LIN {X 0,Y 227.107,Z 476.36,A -85,B 0,C 180,E1 -20579.094,E2 -20579.094} C_VEL
LIN {X 0,Y 226.995,Z 485.322,A -85,B 0,C 180,E1 -20580.664,E2 -20580.664} C_VEL
LIN {X 0,Y 226.013,Z 495.622,A -85,B 0,C 180,E1 -20582.704,E2 -20582.704} C_VEL
LIN {X 0,Y 223.02,Z 505.372,A -85,B 0,C 180,E1 -20584.828,E2 -20584.828} C_VEL
LIN {X 0,Y 220.277,Z 513.339,A -85,B 0,C 180,E1 -20586.998,E2 -20586.998} C_VEL
LIN {X 0,Y 217.787,Z 520.819,A -85,B 0,C 180,E1 -20589.579,E2 -20589.579} C_VEL
LIN {X 0,Y 215.866,Z 526.381,A -85,B 0,C 180,E1 -20591.988,E2 -20591.988} C_VEL
LIN {X 0,Y 214.036,Z 531.459,A -85,B 0,C 180,E1 -20594.775,E2 -20594.775} C_VEL
LIN {X 0,Y 212.725,Z 535.379,A -85,B 0,C 180,E1 -20597.604,E2 -20597.604} C_VEL
LIN {X 0,Y 211.981,Z 538.249,A -85,B 0,C 180,E1 -20600.463,E2 -20600.463} C_VEL
LIN {X 0,Y 211.672,Z 539.61,A -85,B 0,C 180,E1 -20602.373,E2 -20602.373} C_VEL
LIN {X 0,Y 211.57,Z 541.409,A -85,B 0,C 180,E1 -20604.285,E2 -20604.285} C_VEL
LIN {X 0,Y 211.515,Z 543.682,A -85,B 0,C 180,E1 -20606.194,E2 -20606.194} C_VEL
LIN {X 0,Y 211.604,Z 545.507,A -85,B 0,C 180,E1 -20608.101,E2 -20608.101} C_VEL
LIN {X 0,Y 211.672,Z 546.833,A -85,B 0,C 180,E1 -20610.004,E2 -20610.004} C_VEL
LIN {X 0,Y 211.55,Z 547.738,A -85,B 0,C 180,E1 -20611.908,E2 -20611.908} C_VEL
LIN {X 0,Y 211.496,Z 548.371,A -85,B 0,C 180,E1 -20615.725,E2 -20615.725} C_VEL
LIN {X 0,Y 212.119,Z 547.382,A -85,B 0,C 180,E1 -20619.54,E2 -20619.54} C_VEL
LIN {X 0,Y 213.535,Z 544.883,A -85,B 0,C 180,E1 -20623.324,E2 -20623.324} C_VEL
LIN {X 0,Y 215.163,Z 541.937,A -85,B 0,C 180,E1 -20626.123,E2 -20626.123} C_VEL
LIN {X 0,Y 217.434,Z 538.014,A -85,B 0,C 180,E1 -20628.862,E2 -20628.862} C_VEL
LIN {X 0,Y 220.15,Z 533.028,A -85,B 0,C 180,E1 -20631.542,E2 -20631.542} C_VEL
LIN {X 0,Y 223.777,Z 525.758,A -85,B 0,C 180,E1 -20634.594,E2 -20634.594} C_VEL
LIN {X 0,Y 227.652,Z 518.001,A -85,B 0,C 180,E1 -20637.092,E2 -20637.092} C_VEL
LIN {X 0,Y 231.21,Z 510.223,A -85,B 0,C 180,E1 -20639.104,E2 -20639.104} C_VEL
LIN {X 0,Y 234.36,Z 502.894,A -85,B 0,C 180,E1 -20640.654,E2 -20640.654} C_VEL
LIN {X 0,Y 236.711,Z 492.801,A -85,B 0,C 180,E1 -20642.823,E2 -20642.823} C_VEL
LIN {X 0,Y 238.09,Z 482.378,A -85,B 0,C 180,E1 -20644.888,E2 -20644.888} C_VEL
LIN {X 0,Y 238.492,Z 473.335,A -85,B 0,C 180,E1 -20646.63,E2 -20646.63} C_VEL
LIN {X 0,Y 238.102,Z 467.173,A -85,B 0,C 180,E1 -20647.913,E2 -20647.913} C_VEL
LIN {X 0,Y 237.355,Z 464.057,A -85,B 0,C 180,E1 -20648.702,E2 -20648.702} C_VEL
LIN {X 0,Y 234.077,Z 456.011,A -85,B 0,C 180,E1 -20651.356,E2 -20651.356} C_VEL
LIN {X 0,Y 231.692,Z 450.913,A -85,B 0,C 180,E1 -20653.28,E2 -20653.28} C_VEL
LIN {X 0,Y 229.388,Z 446.355,A -85,B 0,C 180,E1 -20655.196,E2 -20655.196} C_VEL
LIN {X 0,Y 225.763,Z 440.725,A -85,B 0,C 180,E1 -20658.495,E2 -20658.495} C_VEL
LIN {X 0,Y 221.458,Z 435.556,A -85,B 0,C 180,E1 -20663.903,E2 -20663.903} C_VEL
LIN {X 0,Y 220.385,Z 433.781,A -85,B 0,C 180,E1 -20666.703,E2 -20666.703} C_VEL
LIN {X 0,Y 219.942,Z 433.291,A -85,B 0,C 180,E1 -20671.359,E2 -20671.359} C_VEL
LIN {X 0,Y 219.974,Z 433.672,A -85,B 0,C 180,E1 -20673.851,E2 -20673.851} C_VEL
LIN {X 0,Y 222.619,Z 437.606,A -85,B 0,C 180,E1 -20679.496,E2 -20679.496} C_VEL
LIN {X 0,Y 224.538,Z 439.728,A -85,B 0,C 180,E1 -20681.818,E2 -20681.818} C_VEL
LIN {X 0,Y 226.805,Z 443.671,A -85,B 0,C 180,E1 -20684.355,E2 -20684.355} C_VEL
LIN {X 0,Y 228.179,Z 445.399,A -85,B 0,C 180,E1 -20685.527,E2 -20685.527} C_VEL
LIN {X 0,Y 231.264,Z 451.056,A -85,B 0,C 180,E1 -20688.299,E2 -20688.299} C_VEL
LIN {X 0,Y 234.016,Z 457.009,A -85,B 0,C 180,E1 -20690.724,E2 -20690.724} C_VEL
LIN {X 0,Y 235.387,Z 461.443,A -85,B 0,C 180,E1 -20692.134,E2 -20692.134} C_VEL
LIN {X 0,Y 236.792,Z 470.013,A -85,B 0,C 180,E1 -20694.466,E2 -20694.466} C_VEL
LIN {X 0,Y 237.694,Z 479.754,A -85,B 0,C 180,E1 -20697.033,E2 -20697.033} C_VEL
LIN {X 0,Y 237.495,Z 488.082,A -85,B 0,C 180,E1 -20699.152,E2 -20699.152} C_VEL
LIN {X 0,Y 237.09,Z 491.443,A -85,B 0,C 180,E1 -20699.999,E2 -20699.999} C_VEL
LIN {X 0,Y 232.908,Z 501.539,A -85,B 0,C 180,E1 -20702.155,E2 -20702.155} C_VEL
LIN {X 0,Y 228.956,Z 509.883,A -85,B 0,C 180,E1 -20704.401,E2 -20704.401} C_VEL
LIN {X 0,Y 224.768,Z 518.061,A -85,B 0,C 180,E1 -20707.184,E2 -20707.184} C_VEL
LIN {X 0,Y 221.27,Z 524.41,A -85,B 0,C 180,E1 -20710.045,E2 -20710.045} C_VEL
LIN {X 0,Y 218.193,Z 529.458,A -85,B 0,C 180,E1 -20713.03,E2 -20713.03} C_VEL
LIN {X 0,Y 215.768,Z 533.215,A -85,B 0,C 180,E1 -20716.072,E2 -20716.072} C_VEL
LIN {X 0,Y 213.884,Z 535.823,A -85,B 0,C 180,E1 -20719.182,E2 -20719.182} C_VEL
LIN {X 0,Y 212.588,Z 537.273,A -85,B 0,C 180,E1 -20722.224,E2 -20722.224} C_VEL
LIN {X 0,Y 211.491,Z 537.624,A -85,B 0,C 180,E1 -20726.197,E2 -20726.197} C_VEL
LIN {X 0,Y 211.054,Z 536.388,A -85,B 0,C 180,E1 -20730.021,E2 -20730.021} C_VEL
LIN {X 0,Y 211.142,Z 533.636,A -85,B 0,C 180,E1 -20733.675,E2 -20733.675} C_VEL
LIN {X 0,Y 211.606,Z 529.586,A -85,B 0,C 180,E1 -20737.141,E2 -20737.141} C_VEL
LIN {X 0,Y 212.3,Z 524.246,A -85,B 0,C 180,E1 -20740.408,E2 -20740.408} C_VEL
LIN {X 0,Y 213.385,Z 517.047,A -85,B 0,C 180,E1 -20743.76,E2 -20743.76} C_VEL
LIN {X 0,Y 214.635,Z 509.377,A -85,B 0,C 180,E1 -20746.553,E2 -20746.553} C_VEL
LIN {X 0,Y 216.098,Z 501.03,A -85,B 0,C 180,E1 -20749.01,E2 -20749.01} C_VEL
LIN {X 0,Y 217.869,Z 490.887,A -85,B 0,C 180,E1 -20751.429,E2 -20751.429} C_VEL
LIN {X 0,Y 219.678,Z 480.049,A -85,B 0,C 180,E1 -20753.484,E2 -20753.484} C_VEL
LIN {X 0,Y 220.631,Z 473.975,A -85,B 0,C 180,E1 -20754.451,E2 -20754.451} C_VEL
LIN {X 0,Y 219.521,Z 463.198,A -85,B 0,C 180,E1 -20756.089,E2 -20756.089} C_VEL
LIN {X 0,Y 217.827,Z 451.567,A -85,B 0,C 180,E1 -20757.558,E2 -20757.558} C_VEL
LIN {X 0,Y 215.353,Z 437.49,A -85,B 0,C 180,E1 -20758.962,E2 -20758.962} C_VEL
LIN {X 0,Y 213.882,Z 430.023,A -85,B 0,C 180,E1 -20759.573,E2 -20759.573} C_VEL
LIN {X 0,Y 214.408,Z 424.31,A -85,B 0,C 180,E1 -20763.732,E2 -20763.732} C_VEL
LIN {X 0,Y 214.842,Z 420,A -85,B 0,C 180,E1 -20766.883,E2 -20766.883} C_VEL
LIN {X 0,Y 214.392,Z 416.106,A -85,B 0,C 180,E1 -20769.863,E2 -20769.863} C_VEL
LIN {X 0,Y 213.959,Z 413.834,A -85,B 0,C 180,E1 -20771.68,E2 -20771.68} C_VEL
LIN {X 0,Y 213.955,Z 413.836,A -85,B 0,C 180,E1 -20776.703,E2 -20776.703} C_VEL
LIN {X 0,Y 214.178,Z 413.969,A -85,B 0,C 180,E1 -20780.791,E2 -20780.791} C_VEL
LIN {X 0,Y 214.6,Z 417.016,A -85,B 0,C 180,E1 -20784.358,E2 -20784.358} C_VEL
LIN {X 0,Y 215.315,Z 420.362,A -85,B 0,C 180,E1 -20788.125,E2 -20788.125} C_VEL
LIN {X 0,Y 214.618,Z 424.04,A -85,B 0,C 180,E1 -20791.872,E2 -20791.872} C_VEL
LIN {X 0,Y 213.861,Z 428.966,A -85,B 0,C 180,E1 -20796.778,E2 -20796.778} C_VEL
LIN {X 0,Y 216.87,Z 442.299,A -85,B 0,C 180,E1 -20798.146,E2 -20798.146} C_VEL
LIN {X 0,Y 218.947,Z 454.169,A -85,B 0,C 180,E1 -20799.697,E2 -20799.697} C_VEL
LIN {X 0,Y 220.145,Z 464.096,A -85,B 0,C 180,E1 -20801.272,E2 -20801.272} C_VEL
LIN {X 0,Y 220.373,Z 469.215,A -85,B 0,C 180,E1 -20802.193,E2 -20802.193} C_VEL
LIN {X 0,Y 218.765,Z 478.309,A -85,B 0,C 180,E1 -20803.938,E2 -20803.938} C_VEL
LIN {X 0,Y 217.225,Z 486.723,A -85,B 0,C 180,E1 -20805.958,E2 -20805.958} C_VEL
LIN {X 0,Y 215.572,Z 494.91,A -85,B 0,C 180,E1 -20808.437,E2 -20808.437} C_VEL
LIN {X 0,Y 214.193,Z 501.913,A -85,B 0,C 180,E1 -20811.152,E2 -20811.152} C_VEL
LIN {X 0,Y 213.305,Z 506.293,A -85,B 0,C 180,E1 -20813.284,E2 -20813.284} C_VEL
LIN {X 0,Y 212.647,Z 509.865,A -85,B 0,C 180,E1 -20815.44,E2 -20815.44} C_VEL
LIN {X 0,Y 211.937,Z 513.853,A -85,B 0,C 180,E1 -20818.734,E2 -20818.734} C_VEL
LIN {X 0,Y 211.734,Z 515.256,A -85,B 0,C 180,E1 -20820.345,E2 -20820.345} C_VEL
LIN {X 0,Y 211.623,Z 516.355,A -85,B 0,C 180,E1 -20822.092,E2 -20822.092} C_VEL
LIN {X 0,Y 211.682,Z 517.207,A -85,B 0,C 180,E1 -20824.356,E2 -20824.356} C_VEL
LIN {X 0,Y 212.095,Z 517.294,A -85,B 0,C 180,E1 -20827.321,E2 -20827.321} C_VEL
LIN {X 0,Y 213.026,Z 516.046,A -85,B 0,C 180,E1 -20830.642,E2 -20830.642} C_VEL
LIN {X 0,Y 214.453,Z 513.396,A -85,B 0,C 180,E1 -20833.866,E2 -20833.866} C_VEL
LIN {X 0,Y 216.211,Z 509.41,A -85,B 0,C 180,E1 -20836.953,E2 -20836.953} C_VEL
LIN {X 0,Y 218.517,Z 503.868,A -85,B 0,C 180,E1 -20839.967,E2 -20839.967} C_VEL
LIN {X 0,Y 221.065,Z 497.333,A -85,B 0,C 180,E1 -20842.627,E2 -20842.627} C_VEL
LIN {X 0,Y 223.58,Z 490.395,A -85,B 0,C 180,E1 -20844.805,E2 -20844.805} C_VEL
LIN {X 0,Y 226.376,Z 481.786,A -85,B 0,C 180,E1 -20846.945,E2 -20846.945} C_VEL
LIN {X 0,Y 227.405,Z 478.157,A -85,B 0,C 180,E1 -20847.712,E2 -20847.712} C_VEL
LIN {X 0,Y 227.286,Z 469.609,A -85,B 0,C 180,E1 -20849.685,E2 -20849.685} C_VEL
LIN {X 0,Y 226.105,Z 460.131,A -85,B 0,C 180,E1 -20851.706,E2 -20851.706} C_VEL
LIN {X 0,Y 223.465,Z 449.533,A -85,B 0,C 180,E1 -20853.878,E2 -20853.878} C_VEL
LIN {X 0,Y 219.612,Z 438.719,A -85,B 0,C 180,E1 -20856.04,E2 -20856.04} C_VEL
LIN {X 0,Y 217.821,Z 434.765,A -85,B 0,C 180,E1 -20856.863,E2 -20856.863} C_VEL
LIN {X 0,Y 216.374,Z 431.502,A -85,B 0,C 180,E1 -20857.502,E2 -20857.502} C_VEL
LIN {X 0,Y 216.279,Z 430.843,A -85,B 0,C 180,E1 -20857.68,E2 -20857.68} C_VEL
LIN {X 0,Y 216.393,Z 428.394,A -85,B 0,C 180,E1 -20861.048,E2 -20861.048} C_VEL
LIN {X 0,Y 216.088,Z 425.902,A -85,B 0,C 180,E1 -20864.919,E2 -20864.919} C_VEL
LIN {X 0,Y 215.927,Z 423.699,A -85,B 0,C 180,E1 -20868.739,E2 -20868.739} C_VEL
LIN {X 0,Y 215.778,Z 421.782,A -85,B 0,C 180,E1 -20872.515,E2 -20872.515} C_VEL
LIN {X 0,Y 215.579,Z 419.442,A -85,B 0,C 180,E1 -20878.132,E2 -20878.132} C_VEL
LIN {X 0,Y 215.603,Z 418.805,A -85,B 0,C 180,E1 -20880.001,E2 -20880.001} C_VEL
LIN {X 0,Y 215.098,Z 417.933,A -85,B 0,C 180,E1 -20883.747,E2 -20883.747} C_VEL
LIN {X 0,Y 214.973,Z 417.288,A -85,B 0,C 180,E1 -20887.515,E2 -20887.515} C_VEL
LIN {X 0,Y 214.712,Z 417.067,A -85,B 0,C 180,E1 -20891.327,E2 -20891.327} C_VEL
LIN {X 0,Y 214.666,Z 417.171,A -85,B 0,C 180,E1 -20895.184,E2 -20895.184} C_VEL
LIN {X 0,Y 214.684,Z 417.679,A -85,B 0,C 180,E1 -20899.11,E2 -20899.11} C_VEL
LIN {X 0,Y 214.964,Z 418.755,A -85,B 0,C 180,E1 -20903.747,E2 -20903.747} C_VEL
LIN {X 0,Y 215.252,Z 420.378,A -85,B 0,C 180,E1 -20908.181,E2 -20908.181} C_VEL
LIN {X 0,Y 215.658,Z 422.238,A -85,B 0,C 180,E1 -20912.09,E2 -20912.09} C_VEL
LIN {X 0,Y 216.05,Z 424.434,A -85,B 0,C 180,E1 -20915.841,E2 -20915.841} C_VEL
LIN {X 0,Y 216.463,Z 426.44,A -85,B 0,C 180,E1 -20918.819,E2 -20918.819} C_VEL
LIN {X 0,Y 217.088,Z 429.542,A -85,B 0,C 180,E1 -20922.833,E2 -20922.833} C_VEL
LIN {X 0,Y 217.553,Z 431.612,A -85,B 0,C 180,E1 -20925.293,E2 -20925.293} C_VEL
LIN {X 0,Y 218.308,Z 436.035,A -85,B 0,C 180,E1 -20929.926,E2 -20929.926} C_VEL
LIN {X 0,Y 218.922,Z 439.604,A -85,B 0,C 180,E1 -20933.274,E2 -20933.274} C_VEL
LIN {X 0,Y 220.491,Z 443.316,A -85,B 0,C 180,E1 -20933.897,E2 -20933.897} C_VEL
LIN {X 0,Y 221.617,Z 445.206,A -85,B 0,C 180,E1 -20934.292,E2 -20934.292} C_VEL
LIN {X 0,Y 223.284,Z 449.616,A -85,B 0,C 180,E1 -20935.021,E2 -20935.021} C_VEL
LIN {X 0,Y 225.504,Z 459.889,A -85,B 0,C 180,E1 -20936.523,E2 -20936.523} C_VEL
LIN {X 0,Y 226.279,Z 464.944,A -85,B 0,C 180,E1 -20937.292,E2 -20937.292} C_VEL
LIN {X 0,Y 226.13,Z 470.276,A -85,B 0,C 180,E1 -20937.987,E2 -20937.987} C_VEL
LIN {X 0,Y 223.986,Z 479.117,A -85,B 0,C 180,E1 -20939.012,E2 -20939.012} C_VEL
LIN {X 0,Y 221.247,Z 487.606,A -85,B 0,C 180,E1 -20940.16,E2 -20940.16} C_VEL
LIN {X 0,Y 220.192,Z 492.349,A -85,B 0,C 180,E1 -20941.037,E2 -20941.037} C_VEL
LIN {X 0,Y 219.195,Z 498.184,A -85,B 0,C 180,E1 -20942.301,E2 -20942.301} C_VEL
LIN {X 0,Y 216.018,Z 507.395,A -85,B 0,C 180,E1 -20944.469,E2 -20944.469} C_VEL
LIN {X 0,Y 212.766,Z 516.266,A -85,B 0,C 180,E1 -20947.168,E2 -20947.168} C_VEL
LIN {X 0,Y 210.598,Z 522.414,A -85,B 0,C 180,E1 -20949.56,E2 -20949.56} C_VEL
LIN {X 0,Y 208.442,Z 528.143,A -85,B 0,C 180,E1 -20952.34,E2 -20952.34} C_VEL
LIN {X 0,Y 206.595,Z 532.748,A -85,B 0,C 180,E1 -20955.223,E2 -20955.223} C_VEL
LIN {X 0,Y 205.431,Z 536.239,A -85,B 0,C 180,E1 -20958.16,E2 -20958.16} C_VEL
LIN {X 0,Y 204.938,Z 537.978,A -85,B 0,C 180,E1 -20960.132,E2 -20960.132} C_VEL
LIN {X 0,Y 204.49,Z 540.726,A -85,B 0,C 180,E1 -20964.087,E2 -20964.087} C_VEL
LIN {X 0,Y 204.431,Z 543.059,A -85,B 0,C 180,E1 -20966.062,E2 -20966.062} C_VEL
LIN {X 0,Y 204.517,Z 544.953,A -85,B 0,C 180,E1 -20968.035,E2 -20968.035} C_VEL
LIN {X 0,Y 204.607,Z 546.405,A -85,B 0,C 180,E1 -20970.004,E2 -20970.004} C_VEL
LIN {X 0,Y 204.465,Z 547.376,A -85,B 0,C 180,E1 -20971.974,E2 -20971.974} C_VEL
LIN {X 0,Y 204.409,Z 548.15,A -85,B 0,C 180,E1 -20975.925,E2 -20975.925} C_VEL
LIN {X 0,Y 204.655,Z 547.96,A -85,B 0,C 180,E1 -20977.899,E2 -20977.899} C_VEL
LIN {X 0,Y 205.748,Z 546.371,A -85,B 0,C 180,E1 -20981.831,E2 -20981.831} C_VEL
LIN {X 0,Y 207.65,Z 543.268,A -85,B 0,C 180,E1 -20985.714,E2 -20985.714} C_VEL
LIN {X 0,Y 210.743,Z 538.451,A -85,B 0,C 180,E1 -20989.485,E2 -20989.485} C_VEL
LIN {X 0,Y 213.597,Z 533.685,A -85,B 0,C 180,E1 -20992.238,E2 -20992.238} C_VEL
LIN {X 0,Y 217.407,Z 526.705,A -85,B 0,C 180,E1 -20995.365,E2 -20995.365} C_VEL
LIN {X 0,Y 221.447,Z 519.184,A -85,B 0,C 180,E1 -20997.916,E2 -20997.916} C_VEL
LIN {X 0,Y 225.159,Z 511.748,A -85,B 0,C 180,E1 -20999.965,E2 -20999.965} C_VEL
LIN {X 0,Y 228.463,Z 504.778,A -85,B 0,C 180,E1 -21001.534,E2 -21001.534} C_VEL
LIN {X 0,Y 231.081,Z 495.042,A -85,B 0,C 180,E1 -21003.728,E2 -21003.728} C_VEL
LIN {X 0,Y 232.861,Z 484.479,A -85,B 0,C 180,E1 -21005.953,E2 -21005.953} C_VEL
LIN {X 0,Y 233.515,Z 476.733,A -85,B 0,C 180,E1 -21007.543,E2 -21007.543} C_VEL
LIN {X 0,Y 233.359,Z 470.923,A -85,B 0,C 180,E1 -21008.826,E2 -21008.826} C_VEL
LIN {X 0,Y 232.503,Z 467.249,A -85,B 0,C 180,E1 -21009.913,E2 -21009.913} C_VEL
LIN {X 0,Y 229.096,Z 458.34,A -85,B 0,C 180,E1 -21013.164,E2 -21013.164} C_VEL
LIN {X 0,Y 226.729,Z 452.997,A -85,B 0,C 180,E1 -21015.479,E2 -21015.479} C_VEL
LIN {X 0,Y 223.293,Z 447.107,A -85,B 0,C 180,E1 -21019.063,E2 -21019.063} C_VEL
LIN {X 0,Y 219.534,Z 442.158,A -85,B 0,C 180,E1 -21024.387,E2 -21024.387} C_VEL
LIN {X 0,Y 218.629,Z 440.622,A -85,B 0,C 180,E1 -21026.874,E2 -21026.874} C_VEL
LIN {X 0,Y 217.962,Z 440.107,A -85,B 0,C 180,E1 -21031.074,E2 -21031.074} C_VEL
LIN {X 0,Y 218.373,Z 440.693,A -85,B 0,C 180,E1 -21034.01,E2 -21034.01} C_VEL
LIN {X 0,Y 221.232,Z 445.104,A -85,B 0,C 180,E1 -21040.211,E2 -21040.211} C_VEL
LIN {X 0,Y 222.104,Z 446.211,A -85,B 0,C 180,E1 -21041.378,E2 -21041.378} C_VEL
LIN {X 0,Y 225.319,Z 452.004,A -85,B 0,C 180,E1 -21045.234,E2 -21045.234} C_VEL
LIN {X 0,Y 228.051,Z 457.688,A -85,B 0,C 180,E1 -21048.132,E2 -21048.132} C_VEL
LIN {X 0,Y 229.954,Z 462.191,A -85,B 0,C 180,E1 -21050.067,E2 -21050.067} C_VEL
LIN {X 0,Y 231.094,Z 467.143,A -85,B 0,C 180,E1 -21051.719,E2 -21051.719} C_VEL
LIN {X 0,Y 232.005,Z 476.299,A -85,B 0,C 180,E1 -21054.345,E2 -21054.345} C_VEL
LIN {X 0,Y 232.3,Z 484.099,A -85,B 0,C 180,E1 -21056.53,E2 -21056.53} C_VEL
LIN {X 0,Y 231.615,Z 492.033,A -85,B 0,C 180,E1 -21058.695,E2 -21058.695} C_VEL
LIN {X 0,Y 231.279,Z 493.703,A -85,B 0,C 180,E1 -21059.129,E2 -21059.129} C_VEL
LIN {X 0,Y 226.693,Z 503.858,A -85,B 0,C 180,E1 -21061.424,E2 -21061.424} C_VEL
LIN {X 0,Y 222.76,Z 511.567,A -85,B 0,C 180,E1 -21063.617,E2 -21063.617} C_VEL
LIN {X 0,Y 219.069,Z 518.184,A -85,B 0,C 180,E1 -21065.978,E2 -21065.978} C_VEL
LIN {X 0,Y 215.845,Z 523.643,A -85,B 0,C 180,E1 -21068.425,E2 -21068.425} C_VEL
LIN {X 0,Y 212.506,Z 528.882,A -85,B 0,C 180,E1 -21071.445,E2 -21071.445} C_VEL
LIN {X 0,Y 210.126,Z 532.325,A -85,B 0,C 180,E1 -21074.07,E2 -21074.07} C_VEL
LIN {X 0,Y 207.53,Z 535.62,A -85,B 0,C 180,E1 -21077.745,E2 -21077.745} C_VEL
LIN {X 0,Y 206.41,Z 536.885,A -85,B 0,C 180,E1 -21079.906,E2 -21079.906} C_VEL
LIN {X 0,Y 205.38,Z 537.715,A -85,B 0,C 180,E1 -21082.485,E2 -21082.485} C_VEL
LIN {X 0,Y 204.821,Z 537.911,A -85,B 0,C 180,E1 -21084.314,E2 -21084.314} C_VEL
LIN {X 0,Y 204.341,Z 537.691,A -85,B 0,C 180,E1 -21086.583,E2 -21086.583} C_VEL
LIN {X 0,Y 203.93,Z 536.052,A -85,B 0,C 180,E1 -21090.501,E2 -21090.501} C_VEL
LIN {X 0,Y 204.091,Z 533.007,A -85,B 0,C 180,E1 -21094.258,E2 -21094.258} C_VEL
LIN {X 0,Y 204.657,Z 528.56,A -85,B 0,C 180,E1 -21097.825,E2 -21097.825} C_VEL
LIN {X 0,Y 205.389,Z 522.933,A -85,B 0,C 180,E1 -21101.162,E2 -21101.162} C_VEL
LIN {X 0,Y 206.507,Z 515.862,A -85,B 0,C 180,E1 -21104.378,E2 -21104.378} C_VEL
LIN {X 0,Y 207.986,Z 507.205,A -85,B 0,C 180,E1 -21107.478,E2 -21107.478} C_VEL
LIN {X 0,Y 209.636,Z 498.083,A -85,B 0,C 180,E1 -21110.074,E2 -21110.074} C_VEL
LIN {X 0,Y 211.515,Z 487.513,A -85,B 0,C 180,E1 -21112.493,E2 -21112.493} C_VEL
LIN {X 0,Y 213.48,Z 475.762,A -85,B 0,C 180,E1 -21114.619,E2 -21114.619} C_VEL
LIN {X 0,Y 213.592,Z 472.582,A -85,B 0,C 180,E1 -21115.142,E2 -21115.142} C_VEL
LIN {X 0,Y 211.972,Z 459.691,A -85,B 0,C 180,E1 -21117.078,E2 -21117.078} C_VEL
LIN {X 0,Y 210.033,Z 446.74,A -85,B 0,C 180,E1 -21118.647,E2 -21118.647} C_VEL
LIN {X 0,Y 207.304,Z 432.461,A -85,B 0,C 180,E1 -21119.992,E2 -21119.992} C_VEL
LIN {X 0,Y 206.892,Z 430.14,A -85,B 0,C 180,E1 -21120.207,E2 -21120.207} C_VEL
LIN {X 0,Y 207.572,Z 423.759,A -85,B 0,C 180,E1 -21124.959,E2 -21124.959} C_VEL
LIN {X 0,Y 207.819,Z 420.894,A -85,B 0,C 180,E1 -21127.109,E2 -21127.109} C_VEL
LIN {X 0,Y 207.334,Z 416.981,A -85,B 0,C 180,E1 -21130.182,E2 -21130.182} C_VEL
LIN {X 0,Y 206.933,Z 414.71,A -85,B 0,C 180,E1 -21131.979,E2 -21131.979} C_VEL
LIN {X 0,Y 206.898,Z 414.714,A -85,B 0,C 180,E1 -21136.24,E2 -21136.24} C_VEL
LIN {X 0,Y 207.13,Z 414.879,A -85,B 0,C 180,E1 -21140.228,E2 -21140.228} C_VEL
LIN {X 0,Y 207.441,Z 416.487,A -85,B 0,C 180,E1 -21142.207,E2 -21142.207} C_VEL
LIN {X 0,Y 208.293,Z 421.478,A -85,B 0,C 180,E1 -21148.062,E2 -21148.062} C_VEL
LIN {X 0,Y 207.56,Z 425.216,A -85,B 0,C 180,E1 -21151.936,E2 -21151.936} C_VEL
LIN {X 0,Y 206.908,Z 429.282,A -85,B 0,C 180,E1 -21156.028,E2 -21156.028} C_VEL
LIN {X 0,Y 209.582,Z 440.667,A -85,B 0,C 180,E1 -21157.22,E2 -21157.22} C_VEL
LIN {X 0,Y 211.561,Z 451.316,A -85,B 0,C 180,E1 -21158.593,E2 -21158.593} C_VEL
LIN {X 0,Y 212.946,Z 461.639,A -85,B 0,C 180,E1 -21160.214,E2 -21160.214} C_VEL
LIN {X 0,Y 213.573,Z 469.341,A -85,B 0,C 180,E1 -21161.623,E2 -21161.623} C_VEL
LIN {X 0,Y 211.956,Z 478.435,A -85,B 0,C 180,E1 -21163.416,E2 -21163.416} C_VEL
LIN {X 0,Y 210.337,Z 486.907,A -85,B 0,C 180,E1 -21165.499,E2 -21165.499} C_VEL
LIN {X 0,Y 208.511,Z 495.858,A -85,B 0,C 180,E1 -21168.313,E2 -21168.313} C_VEL
LIN {X 0,Y 207.179,Z 502.172,A -85,B 0,C 180,E1 -21170.861,E2 -21170.861} C_VEL
LIN {X 0,Y 205.918,Z 508.463,A -85,B 0,C 180,E1 -21174.172,E2 -21174.172} C_VEL
LIN {X 0,Y 205.144,Z 512.426,A -85,B 0,C 180,E1 -21177.036,E2 -21177.036} C_VEL
LIN {X 0,Y 204.84,Z 514.193,A -85,B 0,C 180,E1 -21178.702,E2 -21178.702} C_VEL
LIN {X 0,Y 204.582,Z 516.047,A -85,B 0,C 180,E1 -21181.011,E2 -21181.011} C_VEL
LIN {X 0,Y 204.615,Z 517.591,A -85,B 0,C 180,E1 -21184.48,E2 -21184.48} C_VEL
LIN {X 0,Y 205.166,Z 517.634,A -85,B 0,C 180,E1 -21188.061,E2 -21188.061} C_VEL
LIN {X 0,Y 206.229,Z 516.29,A -85,B 0,C 180,E1 -21191.434,E2 -21191.434} C_VEL
LIN {X 0,Y 207.804,Z 513.504,A -85,B 0,C 180,E1 -21194.748,E2 -21194.748} C_VEL
LIN {X 0,Y 209.758,Z 509.404,A -85,B 0,C 180,E1 -21197.926,E2 -21197.926} C_VEL
LIN {X 0,Y 212.22,Z 503.739,A -85,B 0,C 180,E1 -21201.009,E2 -21201.009} C_VEL
LIN {X 0,Y 214.59,Z 498.078,A -85,B 0,C 180,E1 -21203.35,E2 -21203.35} C_VEL
LIN {X 0,Y 217.215,Z 491.248,A -85,B 0,C 180,E1 -21205.585,E2 -21205.585} C_VEL
LIN {X 0,Y 220.509,Z 481.657,A -85,B 0,C 180,E1 -21208.021,E2 -21208.021} C_VEL
LIN {X 0,Y 221.057,Z 479.028,A -85,B 0,C 180,E1 -21208.629,E2 -21208.629} C_VEL
LIN {X 0,Y 221.01,Z 469.827,A -85,B 0,C 180,E1 -21210.862,E2 -21210.862} C_VEL
LIN {X 0,Y 219.794,Z 460.783,A -85,B 0,C 180,E1 -21212.911,E2 -21212.911} C_VEL
LIN {X 0,Y 217.291,Z 450.615,A -85,B 0,C 180,E1 -21215.137,E2 -21215.137} C_VEL
LIN {X 0,Y 213.83,Z 440.763,A -85,B 0,C 180,E1 -21217.284,E2 -21217.284} C_VEL
LIN {X 0,Y 211.283,Z 435.317,A -85,B 0,C 180,E1 -21218.538,E2 -21218.538} C_VEL
LIN {X 0,Y 209.635,Z 432.014,A -85,B 0,C 180,E1 -21219.309,E2 -21219.309} C_VEL
LIN {X 0,Y 209.436,Z 431.215,A -85,B 0,C 180,E1 -21219.49,E2 -21219.49} C_VEL
LIN {X 0,Y 209.411,Z 429.241,A -85,B 0,C 180,E1 -21222.42,E2 -21222.42} C_VEL
LIN {X 0,Y 209.136,Z 426.543,A -85,B 0,C 180,E1 -21227.018,E2 -21227.018} C_VEL
LIN {X 0,Y 209.047,Z 424.805,A -85,B 0,C 180,E1 -21230.324,E2 -21230.324} C_VEL
LIN {X 0,Y 208.824,Z 423.055,A -85,B 0,C 180,E1 -21234.206,E2 -21234.206} C_VEL
LIN {X 0,Y 208.801,Z 421.558,A -85,B 0,C 180,E1 -21238.072,E2 -21238.072} C_VEL
LIN {X 0,Y 208.834,Z 420.952,A -85,B 0,C 180,E1 -21240.001,E2 -21240.001} C_VEL
LIN {X 0,Y 208.337,Z 420.113,A -85,B 0,C 180,E1 -21243.869,E2 -21243.869} C_VEL
LIN {X 0,Y 208.219,Z 419.511,A -85,B 0,C 180,E1 -21247.76,E2 -21247.76} C_VEL
LIN {X 0,Y 207.962,Z 419.339,A -85,B 0,C 180,E1 -21251.7,E2 -21251.7} C_VEL
LIN {X 0,Y 207.954,Z 419.497,A -85,B 0,C 180,E1 -21255.687,E2 -21255.687} C_VEL
LIN {X 0,Y 207.98,Z 420.091,A -85,B 0,C 180,E1 -21259.751,E2 -21259.751} C_VEL
LIN {X 0,Y 208.265,Z 421.234,A -85,B 0,C 180,E1 -21264.352,E2 -21264.352} C_VEL
LIN {X 0,Y 208.543,Z 422.914,A -85,B 0,C 180,E1 -21268.823,E2 -21268.823} C_VEL
LIN {X 0,Y 208.965,Z 424.812,A -85,B 0,C 180,E1 -21272.784,E2 -21272.784} C_VEL
LIN {X 0,Y 209.423,Z 427.415,A -85,B 0,C 180,E1 -21277.162,E2 -21277.162} C_VEL
LIN {X 0,Y 210.113,Z 430.844,A -85,B 0,C 180,E1 -21281.989,E2 -21281.989} C_VEL
LIN {X 0,Y 210.746,Z 433.745,A -85,B 0,C 180,E1 -21285.555,E2 -21285.555} C_VEL
LIN {X 0,Y 211.426,Z 437.734,A -85,B 0,C 180,E1 -21289.867,E2 -21289.867} C_VEL
LIN {X 0,Y 211.648,Z 439.23,A -85,B 0,C 180,E1 -21291.351,E2 -21291.351} C_VEL
LIN {X 0,Y 213.065,Z 442.663,A -85,B 0,C 180,E1 -21291.988,E2 -21291.988} C_VEL
LIN {X 0,Y 214.713,Z 445.314,A -85,B 0,C 180,E1 -21292.623,E2 -21292.623} C_VEL
LIN {X 0,Y 217.817,Z 452.147,A -85,B 0,C 180,E1 -21294.015,E2 -21294.015} C_VEL
LIN {X 0,Y 219.888,Z 462.891,A -85,B 0,C 180,E1 -21295.712,E2 -21295.712} C_VEL
LIN {X 0,Y 220.939,Z 474.182,A -85,B 0,C 180,E1 -21297.594,E2 -21297.594} C_VEL
LIN {X 0,Y 220.86,Z 485.306,A -85,B 0,C 180,E1 -21299.621,E2 -21299.621} C_VEL
LIN {X 0,Y 220.192,Z 492.349,A -85,B 0,C 180,E1 -21301.037,E2 -21301.037} C_VEL
LIN {X 0,Y 219.066,Z 495.489,A -85,B 0,C 180,E1 -21301.6,E2 -21301.6} C_VEL
LIN {X 0,Y 215.326,Z 500.394,A -85,B 0,C 180,E1 -21302.295,E2 -21302.295} C_VEL
LIN {X 0,Y 211.217,Z 505.108,A -85,B 0,C 180,E1 -21303.043,E2 -21303.043} C_VEL
LIN {X 0,Y 209.564,Z 507.881,A -85,B 0,C 180,E1 -21303.697,E2 -21303.697} C_VEL
LIN {X 0,Y 206.218,Z 516.426,A -85,B 0,C 180,E1 -21306.399,E2 -21306.399} C_VEL
LIN {X 0,Y 203.669,Z 523.161,A -85,B 0,C 180,E1 -21309.179,E2 -21309.179} C_VEL
LIN {X 0,Y 201.634,Z 528.097,A -85,B 0,C 180,E1 -21311.723,E2 -21311.723} C_VEL
LIN {X 0,Y 199.711,Z 532.601,A -85,B 0,C 180,E1 -21314.702,E2 -21314.702} C_VEL
LIN {X 0,Y 198.455,Z 536.01,A -85,B 0,C 180,E1 -21317.737,E2 -21317.737} C_VEL
LIN {X 0,Y 197.565,Z 539.01,A -85,B 0,C 180,E1 -21321.824,E2 -21321.824} C_VEL
LIN {X 0,Y 197.446,Z 539.975,A -85,B 0,C 180,E1 -21323.875,E2 -21323.875} C_VEL
LIN {X 0,Y 197.375,Z 542.43,A -85,B 0,C 180,E1 -21325.921,E2 -21325.921} C_VEL
LIN {X 0,Y 197.433,Z 544.392,A -85,B 0,C 180,E1 -21327.965,E2 -21327.965} C_VEL
LIN {X 0,Y 197.543,Z 545.925,A -85,B 0,C 180,E1 -21330.005,E2 -21330.005} C_VEL
LIN {X 0,Y 197.38,Z 547.011,A -85,B 0,C 180,E1 -21332.045,E2 -21332.045} C_VEL
LIN {X 0,Y 197.348,Z 547.915,A -85,B 0,C 180,E1 -21336.137,E2 -21336.137} C_VEL
LIN {X 0,Y 198.084,Z 547.318,A -85,B 0,C 180,E1 -21340.223,E2 -21340.223} C_VEL
LIN {X 0,Y 199.693,Z 545.134,A -85,B 0,C 180,E1 -21344.266,E2 -21344.266} C_VEL
LIN {X 0,Y 201.538,Z 542.507,A -85,B 0,C 180,E1 -21347.246,E2 -21347.246} C_VEL
LIN {X 0,Y 205.036,Z 537.533,A -85,B 0,C 180,E1 -21351.099,E2 -21351.099} C_VEL
LIN {X 0,Y 208.666,Z 531.655,A -85,B 0,C 180,E1 -21354.369,E2 -21354.369} C_VEL
LIN {X 0,Y 213.096,Z 524.206,A -85,B 0,C 180,E1 -21357.503,E2 -21357.503} C_VEL
LIN {X 0,Y 217.524,Z 516.311,A -85,B 0,C 180,E1 -21360.056,E2 -21360.056} C_VEL
LIN {X 0,Y 222.575,Z 506.526,A -85,B 0,C 180,E1 -21362.469,E2 -21362.469} C_VEL
LIN {X 0,Y 225.313,Z 498.034,A -85,B 0,C 180,E1 -21364.507,E2 -21364.507} C_VEL
LIN {X 0,Y 227.338,Z 489.101,A -85,B 0,C 180,E1 -21366.507,E2 -21366.507} C_VEL
LIN {X 0,Y 228.497,Z 480.432,A -85,B 0,C 180,E1 -21368.405,E2 -21368.405} C_VEL
LIN {X 0,Y 228.635,Z 474.645,A -85,B 0,C 180,E1 -21369.782,E2 -21369.782} C_VEL
LIN {X 0,Y 227.84,Z 471.269,A -85,B 0,C 180,E1 -21370.908,E2 -21370.908} C_VEL
LIN {X 0,Y 225.112,Z 463.142,A -85,B 0,C 180,E1 -21374.104,E2 -21374.104} C_VEL
LIN {X 0,Y 223.162,Z 458.308,A -85,B 0,C 180,E1 -21376.418,E2 -21376.418} C_VEL
LIN {X 0,Y 220.824,Z 453.689,A -85,B 0,C 180,E1 -21379.318,E2 -21379.318} C_VEL
LIN {X 0,Y 217.446,Z 448.84,A -85,B 0,C 180,E1 -21384.669,E2 -21384.669} C_VEL
LIN {X 0,Y 216.679,Z 447.414,A -85,B 0,C 180,E1 -21387.089,E2 -21387.089} C_VEL
LIN {X 0,Y 216.099,Z 446.937,A -85,B 0,C 180,E1 -21391.42,E2 -21391.42} C_VEL
LIN {X 0,Y 216.292,Z 447.149,A -85,B 0,C 180,E1 -21392.941,E2 -21392.941} C_VEL
LIN {X 0,Y 216.675,Z 448.308,A -85,B 0,C 180,E1 -21395.264,E2 -21395.264} C_VEL
LIN {X 0,Y 219.169,Z 452.126,A -85,B 0,C 180,E1 -21400.501,E2 -21400.501} C_VEL
LIN {X 0,Y 221.788,Z 457.496,A -85,B 0,C 180,E1 -21404.413,E2 -21404.413} C_VEL
LIN {X 0,Y 224.098,Z 462.725,A -85,B 0,C 180,E1 -21407.318,E2 -21407.318} C_VEL
LIN {X 0,Y 225.632,Z 466.849,A -85,B 0,C 180,E1 -21409.228,E2 -21409.228} C_VEL
LIN {X 0,Y 226.367,Z 470.206,A -85,B 0,C 180,E1 -21410.489,E2 -21410.489} C_VEL
LIN {X 0,Y 226.881,Z 477.91,A -85,B 0,C 180,E1 -21412.882,E2 -21412.882} C_VEL
LIN {X 0,Y 226.88,Z 486.712,A -85,B 0,C 180,E1 -21415.558,E2 -21415.558} C_VEL
LIN {X 0,Y 225.999,Z 494.372,A -85,B 0,C 180,E1 -21417.772,E2 -21417.772} C_VEL
LIN {X 0,Y 224.988,Z 497.22,A -85,B 0,C 180,E1 -21418.456,E2 -21418.456} C_VEL
LIN {X 0,Y 220.001,Z 507.077,A -85,B 0,C 180,E1 -21420.915,E2 -21420.915} C_VEL
LIN {X 0,Y 215.805,Z 514.542,A -85,B 0,C 180,E1 -21423.266,E2 -21423.266} C_VEL
LIN {X 0,Y 211.927,Z 520.874,A -85,B 0,C 180,E1 -21425.779,E2 -21425.779} C_VEL
LIN {X 0,Y 208.137,Z 526.634,A -85,B 0,C 180,E1 -21428.739,E2 -21428.739} C_VEL
LIN {X 0,Y 204.798,Z 531.196,A -85,B 0,C 180,E1 -21431.882,E2 -21431.882} C_VEL
LIN {X 0,Y 202.893,Z 533.628,A -85,B 0,C 180,E1 -21434.083,E2 -21434.083} C_VEL
LIN {X 0,Y 201.325,Z 535.453,A -85,B 0,C 180,E1 -21436.216,E2 -21436.216} C_VEL
LIN {X 0,Y 199.987,Z 536.804,A -85,B 0,C 180,E1 -21438.437,E2 -21438.437} C_VEL
LIN {X 0,Y 198.942,Z 537.707,A -85,B 0,C 180,E1 -21440.687,E2 -21440.687} C_VEL
LIN {X 0,Y 198.099,Z 538.1,A -85,B 0,C 180,E1 -21442.969,E2 -21442.969} C_VEL
LIN {X 0,Y 197.159,Z 537.638,A -85,B 0,C 180,E1 -21446.974,E2 -21446.974} C_VEL
LIN {X 0,Y 196.814,Z 535.642,A -85,B 0,C 180,E1 -21451.011,E2 -21451.011} C_VEL
LIN {X 0,Y 197.064,Z 532.21,A -85,B 0,C 180,E1 -21454.883,E2 -21454.883} C_VEL
LIN {X 0,Y 197.705,Z 527.475,A -85,B 0,C 180,E1 -21458.546,E2 -21458.546} C_VEL
LIN {X 0,Y 198.62,Z 520.938,A -85,B 0,C 180,E1 -21462.244,E2 -21462.244} C_VEL
LIN {X 0,Y 199.733,Z 514.076,A -85,B 0,C 180,E1 -21465.267,E2 -21465.267} C_VEL
LIN {X 0,Y 201.032,Z 506.692,A -85,B 0,C 180,E1 -21467.895,E2 -21467.895} C_VEL
LIN {X 0,Y 202.928,Z 496.553,A -85,B 0,C 180,E1 -21470.792,E2 -21470.792} C_VEL
LIN {X 0,Y 204.662,Z 487.096,A -85,B 0,C 180,E1 -21472.976,E2 -21472.976} C_VEL
LIN {X 0,Y 206.682,Z 475.161,A -85,B 0,C 180,E1 -21475.169,E2 -21475.169} C_VEL
LIN {X 0,Y 205.472,Z 463.298,A -85,B 0,C 180,E1 -21477.108,E2 -21477.108} C_VEL
LIN {X 0,Y 203.609,Z 450.517,A -85,B 0,C 180,E1 -21478.814,E2 -21478.814} C_VEL
LIN {X 0,Y 201.3,Z 437.212,A -85,B 0,C 180,E1 -21480.232,E2 -21480.232} C_VEL
LIN {X 0,Y 199.95,Z 430.28,A -85,B 0,C 180,E1 -21480.856,E2 -21480.856} C_VEL
LIN {X 0,Y 200.631,Z 424.03,A -85,B 0,C 180,E1 -21485.61,E2 -21485.61} C_VEL
LIN {X 0,Y 200.684,Z 420.414,A -85,B 0,C 180,E1 -21488.421,E2 -21488.421} C_VEL
LIN {X 0,Y 199.883,Z 415.588,A -85,B 0,C 180,E1 -21492.441,E2 -21492.441} C_VEL
LIN {X 0,Y 199.881,Z 415.588,A -85,B 0,C 180,E1 -21497.817,E2 -21497.817} C_VEL
LIN {X 0,Y 200.037,Z 415.814,A -85,B 0,C 180,E1 -21499.649,E2 -21499.649} C_VEL
LIN {X 0,Y 200.411,Z 417.603,A -85,B 0,C 180,E1 -21501.932,E2 -21501.932} C_VEL
LIN {X 0,Y 201.29,Z 422.636,A -85,B 0,C 180,E1 -21507.995,E2 -21507.995} C_VEL
LIN {X 0,Y 200.503,Z 426.381,A -85,B 0,C 180,E1 -21512.004,E2 -21512.004} C_VEL
LIN {X 0,Y 199.959,Z 429.566,A -85,B 0,C 180,E1 -21515.226,E2 -21515.226} C_VEL
LIN {X 0,Y 202.676,Z 440.939,A -85,B 0,C 180,E1 -21516.466,E2 -21516.466} C_VEL
LIN {X 0,Y 204.68,Z 451.586,A -85,B 0,C 180,E1 -21517.89,E2 -21517.89} C_VEL
LIN {X 0,Y 206.046,Z 461.884,A -85,B 0,C 180,E1 -21519.567,E2 -21519.567} C_VEL
LIN {X 0,Y 206.765,Z 469.489,A -85,B 0,C 180,E1 -21521.018,E2 -21521.018} C_VEL
LIN {X 0,Y 204.933,Z 479.755,A -85,B 0,C 180,E1 -21523.127,E2 -21523.127} C_VEL
LIN {X 0,Y 203.203,Z 488.402,A -85,B 0,C 180,E1 -21525.397,E2 -21525.397} C_VEL
LIN {X 0,Y 201.649,Z 495.616,A -85,B 0,C 180,E1 -21527.751,E2 -21527.751} C_VEL
LIN {X 0,Y 200.189,Z 502.424,A -85,B 0,C 180,E1 -21530.547,E2 -21530.547} C_VEL
LIN {X 0,Y 199.039,Z 507.74,A -85,B 0,C 180,E1 -21533.359,E2 -21533.359} C_VEL
LIN {X 0,Y 198.216,Z 511.955,A -85,B 0,C 180,E1 -21536.278,E2 -21536.278} C_VEL
LIN {X 0,Y 197.578,Z 515.548,A -85,B 0,C 180,E1 -21539.861,E2 -21539.861} C_VEL
LIN {X 0,Y 197.451,Z 517.105,A -85,B 0,C 180,E1 -21542.263,E2 -21542.263} C_VEL
LIN {X 0,Y 197.57,Z 518.081,A -85,B 0,C 180,E1 -21545.1,E2 -21545.1} C_VEL
LIN {X 0,Y 198.248,Z 518,A -85,B 0,C 180,E1 -21548.748,E2 -21548.748} C_VEL
LIN {X 0,Y 199.451,Z 516.511,A -85,B 0,C 180,E1 -21552.272,E2 -21552.272} C_VEL
LIN {X 0,Y 201.178,Z 513.633,A -85,B 0,C 180,E1 -21555.679,E2 -21555.679} C_VEL
LIN {X 0,Y 203.316,Z 509.391,A -85,B 0,C 180,E1 -21558.947,E2 -21558.947} C_VEL
LIN {X 0,Y 206.048,Z 503.585,A -85,B 0,C 180,E1 -21562.125,E2 -21562.125} C_VEL
LIN {X 0,Y 208.781,Z 497.367,A -85,B 0,C 180,E1 -21564.673,E2 -21564.673} C_VEL
LIN {X 0,Y 212.002,Z 489.236,A -85,B 0,C 180,E1 -21567.257,E2 -21567.257} C_VEL
LIN {X 0,Y 214.742,Z 481.331,A -85,B 0,C 180,E1 -21569.231,E2 -21569.231} C_VEL
LIN {X 0,Y 214.899,Z 471.757,A -85,B 0,C 180,E1 -21571.694,E2 -21571.694} C_VEL
LIN {X 0,Y 213.915,Z 463.384,A -85,B 0,C 180,E1 -21573.743,E2 -21573.743} C_VEL
LIN {X 0,Y 211.725,Z 453.51,A -85,B 0,C 180,E1 -21576.082,E2 -21576.082} C_VEL
LIN {X 0,Y 208.66,Z 444.329,A -85,B 0,C 180,E1 -21578.254,E2 -21578.254} C_VEL
LIN {X 0,Y 206.583,Z 439.696,A -85,B 0,C 180,E1 -21579.442,E2 -21579.442} C_VEL
LIN {X 0,Y 204.702,Z 435.899,A -85,B 0,C 180,E1 -21580.444,E2 -21580.444} C_VEL
LIN {X 0,Y 202.807,Z 432.57,A -85,B 0,C 180,E1 -21581.37,E2 -21581.37} C_VEL
LIN {X 0,Y 202.549,Z 431.544,A -85,B 0,C 180,E1 -21581.608,E2 -21581.608} C_VEL
LIN {X 0,Y 202.299,Z 428.667,A -85,B 0,C 180,E1 -21586.565,E2 -21586.565} C_VEL
LIN {X 0,Y 202.219,Z 426.927,A -85,B 0,C 180,E1 -21589.993,E2 -21589.993} C_VEL
LIN {X 0,Y 202.042,Z 425.177,A -85,B 0,C 180,E1 -21594.011,E2 -21594.011} C_VEL
LIN {X 0,Y 202.026,Z 423.701,A -85,B 0,C 180,E1 -21598.007,E2 -21598.007} C_VEL
LIN {X 0,Y 202.072,Z 423.096,A -85,B 0,C 180,E1 -21600.001,E2 -21600.001} C_VEL
LIN {X 0,Y 201.585,Z 422.294,A -85,B 0,C 180,E1 -21603.999,E2 -21603.999} C_VEL
LIN {X 0,Y 201.466,Z 421.743,A -85,B 0,C 180,E1 -21608.022,E2 -21608.022} C_VEL
LIN {X 0,Y 201.232,Z 421.626,A -85,B 0,C 180,E1 -21612.097,E2 -21612.097} C_VEL
LIN {X 0,Y 201.228,Z 421.859,A -85,B 0,C 180,E1 -21616.225,E2 -21616.225} C_VEL
LIN {X 0,Y 201.296,Z 422.531,A -85,B 0,C 180,E1 -21620.435,E2 -21620.435} C_VEL
LIN {X 0,Y 201.548,Z 423.644,A -85,B 0,C 180,E1 -21624.737,E2 -21624.737} C_VEL
LIN {X 0,Y 201.872,Z 425.447,A -85,B 0,C 180,E1 -21629.512,E2 -21629.512} C_VEL
LIN {X 0,Y 202.26,Z 427.535,A -85,B 0,C 180,E1 -21633.778,E2 -21633.778} C_VEL
LIN {X 0,Y 202.802,Z 430.449,A -85,B 0,C 180,E1 -21638.594,E2 -21638.594} C_VEL
LIN {X 0,Y 203.582,Z 434.124,A -85,B 0,C 180,E1 -21643.665,E2 -21643.665} C_VEL
LIN {X 0,Y 204.246,Z 437.671,A -85,B 0,C 180,E1 -21647.865,E2 -21647.865} C_VEL
LIN {X 0,Y 204.432,Z 438.915,A -85,B 0,C 180,E1 -21649.225,E2 -21649.225} C_VEL
LIN {X 0,Y 205.828,Z 442.202,A -85,B 0,C 180,E1 -21649.912,E2 -21649.912} C_VEL
LIN {X 0,Y 207.555,Z 444.985,A -85,B 0,C 180,E1 -21650.664,E2 -21650.664} C_VEL
LIN {X 0,Y 209.686,Z 448.993,A -85,B 0,C 180,E1 -21651.639,E2 -21651.639} C_VEL
LIN {X 0,Y 212.386,Z 455.155,A -85,B 0,C 180,E1 -21653.009,E2 -21653.009} C_VEL
LIN {X 0,Y 213.966,Z 463.546,A -85,B 0,C 180,E1 -21654.482,E2 -21654.482} C_VEL
LIN {X 0,Y 214.87,Z 473.424,A -85,B 0,C 180,E1 -21656.224,E2 -21656.224} C_VEL
LIN {X 0,Y 214.831,Z 484.235,A -85,B 0,C 180,E1 -21658.275,E2 -21658.275} C_VEL
LIN {X 0,Y 213.742,Z 494.516,A -85,B 0,C 180,E1 -21660.454,E2 -21660.454} C_VEL
LIN {X 0,Y 212.949,Z 498.649,A -85,B 0,C 180,E1 -21661.415,E2 -21661.415} C_VEL
LIN {X 0,Y 209.564,Z 507.881,A -85,B 0,C 180,E1 -21663.697,E2 -21663.697} C_VEL
LIN {X 0,Y 207.467,Z 511.83,A -85,B 0,C 180,E1 -21664.773,E2 -21664.773} C_VEL
LIN {X 0,Y 202.533,Z 517.782,A -85,B 0,C 180,E1 -21666.509,E2 -21666.509} C_VEL
LIN {X 0,Y 197.697,Z 523.073,A -85,B 0,C 180,E1 -21668.456,E2 -21668.456} C_VEL
LIN {X 0,Y 195.789,Z 525.9,A -85,B 0,C 180,E1 -21669.843,E2 -21669.843} C_VEL
LIN {X 0,Y 193.475,Z 531.115,A -85,B 0,C 180,E1 -21673.111,E2 -21673.111} C_VEL
LIN {X 0,Y 191.822,Z 534.805,A -85,B 0,C 180,E1 -21676.228,E2 -21676.228} C_VEL
LIN {X 0,Y 190.884,Z 537.461,A -85,B 0,C 180,E1 -21679.397,E2 -21679.397} C_VEL
LIN {X 0,Y 190.51,Z 538.703,A -85,B 0,C 180,E1 -21681.519,E2 -21681.519} C_VEL
LIN {X 0,Y 190.361,Z 539.722,A -85,B 0,C 180,E1 -21684.045,E2 -21684.045} C_VEL
LIN {X 0,Y 190.285,Z 542.852,A -85,B 0,C 180,E1 -21686.856,E2 -21686.856} C_VEL
LIN {X 0,Y 190.479,Z 545.409,A -85,B 0,C 180,E1 -21690.005,E2 -21690.005} C_VEL
LIN {X 0,Y 190.185,Z 547.204,A -85,B 0,C 180,E1 -21693.838,E2 -21693.838} C_VEL
LIN {X 0,Y 190.285,Z 547.679,A -85,B 0,C 180,E1 -21696.366,E2 -21696.366} C_VEL
LIN {X 0,Y 191.079,Z 547.23,A -85,B 0,C 180,E1 -21700.602,E2 -21700.602} C_VEL
LIN {X 0,Y 192.788,Z 545.292,A -85,B 0,C 180,E1 -21704.789,E2 -21704.789} C_VEL
LIN {X 0,Y 193.997,Z 543.722,A -85,B 0,C 180,E1 -21706.852,E2 -21706.852} C_VEL
LIN {X 0,Y 197.451,Z 539.395,A -85,B 0,C 180,E1 -21710.855,E2 -21710.855} C_VEL
LIN {X 0,Y 200.604,Z 535.025,A -85,B 0,C 180,E1 -21713.763,E2 -21713.763} C_VEL
LIN {X 0,Y 204.795,Z 528.572,A -85,B 0,C 180,E1 -21717.05,E2 -21717.05} C_VEL
LIN {X 0,Y 209.947,Z 520.353,A -85,B 0,C 180,E1 -21720.145,E2 -21720.145} C_VEL
LIN {X 0,Y 214.957,Z 511.708,A -85,B 0,C 180,E1 -21722.651,E2 -21722.651} C_VEL
LIN {X 0,Y 217.594,Z 506.66,A -85,B 0,C 180,E1 -21723.863,E2 -21723.863} C_VEL
LIN {X 0,Y 220.766,Z 496.985,A -85,B 0,C 180,E1 -21726.276,E2 -21726.276} C_VEL
LIN {X 0,Y 223.148,Z 486.446,A -85,B 0,C 180,E1 -21728.756,E2 -21728.756} C_VEL
LIN {X 0,Y 223.854,Z 480.051,A -85,B 0,C 180,E1 -21730.302,E2 -21730.302} C_VEL
LIN {X 0,Y 223.714,Z 477.458,A -85,B 0,C 180,E1 -21731.064,E2 -21731.064} C_VEL
LIN {X 0,Y 221.603,Z 469.687,A -85,B 0,C 180,E1 -21734.248,E2 -21734.248} C_VEL
LIN {X 0,Y 220.072,Z 464.899,A -85,B 0,C 180,E1 -21736.562,E2 -21736.562} C_VEL
LIN {X 0,Y 217.847,Z 459.905,A -85,B 0,C 180,E1 -21739.817,E2 -21739.817} C_VEL
LIN {X 0,Y 215.079,Z 455.539,A -85,B 0,C 180,E1 -21744.782,E2 -21744.782} C_VEL
LIN {X 0,Y 214.678,Z 454.668,A -85,B 0,C 180,E1 -21746.183,E2 -21746.183} C_VEL
LIN {X 0,Y 214.103,Z 453.854,A -85,B 0,C 180,E1 -21748.595,E2 -21748.595} C_VEL
LIN {X 0,Y 214.006,Z 453.808,A -85,B 0,C 180,E1 -21752.628,E2 -21752.628} C_VEL
LIN {X 0,Y 214.613,Z 455.895,A -85,B 0,C 180,E1 -21756.488,E2 -21756.488} C_VEL
LIN {X 0,Y 216.401,Z 458.742,A -85,B 0,C 180,E1 -21760.369,E2 -21760.369} C_VEL
LIN {X 0,Y 218.738,Z 464.464,A -85,B 0,C 180,E1 -21764.567,E2 -21764.567} C_VEL
LIN {X 0,Y 220.398,Z 468.927,A -85,B 0,C 180,E1 -21767.101,E2 -21767.101} C_VEL
LIN {X 0,Y 221.55,Z 472.95,A -85,B 0,C 180,E1 -21769.027,E2 -21769.027} C_VEL
LIN {X 0,Y 221.948,Z 478.176,A -85,B 0,C 180,E1 -21770.89,E2 -21770.89} C_VEL
LIN {X 0,Y 221.671,Z 488.041,A -85,B 0,C 180,E1 -21774.085,E2 -21774.085} C_VEL
LIN {X 0,Y 220.706,Z 495.198,A -85,B 0,C 180,E1 -21776.348,E2 -21776.348} C_VEL
LIN {X 0,Y 220.074,Z 497.814,A -85,B 0,C 180,E1 -21777.119,E2 -21777.119} C_VEL
LIN {X 0,Y 214.981,Z 507.375,A -85,B 0,C 180,E1 -21779.531,E2 -21779.531} C_VEL
LIN {X 0,Y 210.503,Z 514.813,A -85,B 0,C 180,E1 -21781.913,E2 -21781.913} C_VEL
LIN {X 0,Y 205.979,Z 521.649,A -85,B 0,C 180,E1 -21784.716,E2 -21784.716} C_VEL
LIN {X 0,Y 201.624,Z 527.703,A -85,B 0,C 180,E1 -21788.014,E2 -21788.014} C_VEL
LIN {X 0,Y 198.136,Z 532.065,A -85,B 0,C 180,E1 -21791.249,E2 -21791.249} C_VEL
LIN {X 0,Y 195.27,Z 535.229,A -85,B 0,C 180,E1 -21794.592,E2 -21794.592} C_VEL
LIN {X 0,Y 192.763,Z 537.515,A -85,B 0,C 180,E1 -21798.559,E2 -21798.559} C_VEL
LIN {X 0,Y 191.466,Z 538.277,A -85,B 0,C 180,E1 -21801.534,E2 -21801.534} C_VEL
LIN {X 0,Y 190.693,Z 538.305,A -85,B 0,C 180,E1 -21803.916,E2 -21803.916} C_VEL
LIN {X 0,Y 190.003,Z 537.488,A -85,B 0,C 180,E1 -21807.402,E2 -21807.402} C_VEL
LIN {X 0,Y 189.726,Z 535.13,A -85,B 0,C 180,E1 -21811.565,E2 -21811.565} C_VEL
LIN {X 0,Y 190.068,Z 531.322,A -85,B 0,C 180,E1 -21815.557,E2 -21815.557} C_VEL
LIN {X 0,Y 190.738,Z 526.237,A -85,B 0,C 180,E1 -21819.3,E2 -21819.3} C_VEL
LIN {X 0,Y 191.687,Z 519.89,A -85,B 0,C 180,E1 -21822.833,E2 -21822.833} C_VEL
LIN {X 0,Y 193.008,Z 512.05,A -85,B 0,C 180,E1 -21826.219,E2 -21826.219} C_VEL
LIN {X 0,Y 194.68,Z 503.083,A -85,B 0,C 180,E1 -21829.296,E2 -21829.296} C_VEL
LIN {X 0,Y 196.504,Z 493.615,A -85,B 0,C 180,E1 -21831.889,E2 -21831.889} C_VEL
LIN {X 0,Y 198.429,Z 483.086,A -85,B 0,C 180,E1 -21834.223,E2 -21834.223} C_VEL
LIN {X 0,Y 199.726,Z 474.774,A -85,B 0,C 180,E1 -21835.731,E2 -21835.731} C_VEL
LIN {X 0,Y 198.468,Z 463.695,A -85,B 0,C 180,E1 -21837.611,E2 -21837.611} C_VEL
LIN {X 0,Y 196.57,Z 450.111,A -85,B 0,C 180,E1 -21839.47,E2 -21839.47} C_VEL
LIN {X 0,Y 194.099,Z 436.43,A -85,B 0,C 180,E1 -21840.955,E2 -21840.955} C_VEL
LIN {X 0,Y 192.989,Z 430.405,A -85,B 0,C 180,E1 -21841.525,E2 -21841.525} C_VEL
LIN {X 0,Y 193.705,Z 424.094,A -85,B 0,C 180,E1 -21846.474,E2 -21846.474} C_VEL
LIN {X 0,Y 193.647,Z 421.287,A -85,B 0,C 180,E1 -21848.715,E2 -21848.715} C_VEL
LIN {X 0,Y 192.832,Z 416.465,A -85,B 0,C 180,E1 -21852.822,E2 -21852.822} C_VEL
LIN {X 0,Y 192.883,Z 416.552,A -85,B 0,C 180,E1 -21858.729,E2 -21858.729} C_VEL
LIN {X 0,Y 193.376,Z 418.718,A -85,B 0,C 180,E1 -21861.637,E2 -21861.637} C_VEL
LIN {X 0,Y 193.92,Z 422.059,A -85,B 0,C 180,E1 -21865.839,E2 -21865.839} C_VEL
LIN {X 0,Y 194.283,Z 423.781,A -85,B 0,C 180,E1 -21867.922,E2 -21867.922} C_VEL
LIN {X 0,Y 193.445,Z 427.546,A -85,B 0,C 180,E1 -21872.077,E2 -21872.077} C_VEL
LIN {X 0,Y 193.052,Z 429.85,A -85,B 0,C 180,E1 -21874.367,E2 -21874.367} C_VEL
LIN {X 0,Y 196.012,Z 442.051,A -85,B 0,C 180,E1 -21875.783,E2 -21875.783} C_VEL
LIN {X 0,Y 198.022,Z 453.27,A -85,B 0,C 180,E1 -21877.387,E2 -21877.387} C_VEL
LIN {X 0,Y 199.445,Z 464.71,A -85,B 0,C 180,E1 -21879.375,E2 -21879.375} C_VEL
LIN {X 0,Y 199.905,Z 470.866,A -85,B 0,C 180,E1 -21880.631,E2 -21880.631} C_VEL
LIN {X 0,Y 197.907,Z 480.972,A -85,B 0,C 180,E1 -21882.819,E2 -21882.819} C_VEL
LIN {X 0,Y 196.124,Z 489.453,A -85,B 0,C 180,E1 -21885.165,E2 -21885.165} C_VEL
LIN {X 0,Y 194.421,Z 497.28,A -85,B 0,C 180,E1 -21887.889,E2 -21887.889} C_VEL
LIN {X 0,Y 192.915,Z 503.867,A -85,B 0,C 180,E1 -21890.827,E2 -21890.827} C_VEL
LIN {X 0,Y 191.802,Z 509.003,A -85,B 0,C 180,E1 -21893.764,E2 -21893.764} C_VEL
LIN {X 0,Y 191.126,Z 512.269,A -85,B 0,C 180,E1 -21896.178,E2 -21896.178} C_VEL
LIN {X 0,Y 190.664,Z 514.838,A -85,B 0,C 180,E1 -21898.626,E2 -21898.626} C_VEL
LIN {X 0,Y 190.357,Z 517.204,A -85,B 0,C 180,E1 -21901.881,E2 -21901.881} C_VEL
LIN {X 0,Y 190.368,Z 518.011,A -85,B 0,C 180,E1 -21903.619,E2 -21903.619} C_VEL
LIN {X 0,Y 190.616,Z 518.586,A -85,B 0,C 180,E1 -21906.144,E2 -21906.144} C_VEL
LIN {X 0,Y 191.356,Z 518.36,A -85,B 0,C 180,E1 -21909.533,E2 -21909.533} C_VEL
LIN {X 0,Y 192.727,Z 516.723,A -85,B 0,C 180,E1 -21913.171,E2 -21913.171} C_VEL
LIN {X 0,Y 194.61,Z 513.771,A -85,B 0,C 180,E1 -21916.675,E2 -21916.675} C_VEL
LIN {X 0,Y 196.948,Z 509.408,A -85,B 0,C 180,E1 -21920.036,E2 -21920.036} C_VEL
LIN {X 0,Y 199.936,Z 503.466,A -85,B 0,C 180,E1 -21923.305,E2 -21923.305} C_VEL
LIN {X 0,Y 203.149,Z 496.525,A -85,B 0,C 180,E1 -21926.118,E2 -21926.118} C_VEL
LIN {X 0,Y 206.184,Z 489.205,A -85,B 0,C 180,E1 -21928.436,E2 -21928.436} C_VEL
LIN {X 0,Y 208.275,Z 483.634,A -85,B 0,C 180,E1 -21929.868,E2 -21929.868} C_VEL
LIN {X 0,Y 208.863,Z 476.263,A -85,B 0,C 180,E1 -21931.896,E2 -21931.896} C_VEL
LIN {X 0,Y 208.401,Z 468.353,A -85,B 0,C 180,E1 -21933.999,E2 -21933.999} C_VEL
LIN {X 0,Y 206.801,Z 458.985,A -85,B 0,C 180,E1 -21936.401,E2 -21936.401} C_VEL
LIN {X 0,Y 204.218,Z 449.693,A -85,B 0,C 180,E1 -21938.779,E2 -21938.779} C_VEL
LIN {X 0,Y 201.148,Z 442.352,A -85,B 0,C 180,E1 -21940.806,E2 -21940.806} C_VEL
LIN {X 0,Y 198.209,Z 436.706,A -85,B 0,C 180,E1 -21942.526,E2 -21942.526} C_VEL
LIN {X 0,Y 196.248,Z 433.878,A -85,B 0,C 180,E1 -21943.553,E2 -21943.553} C_VEL
LIN {X 0,Y 195.578,Z 431.878,A -85,B 0,C 180,E1 -21944.098,E2 -21944.098} C_VEL
LIN {X 0,Y 195.449,Z 430.07,A -85,B 0,C 180,E1 -21947.541,E2 -21947.541} C_VEL
LIN {X 0,Y 195.342,Z 428.128,A -85,B 0,C 180,E1 -21951.726,E2 -21951.726} C_VEL
LIN {X 0,Y 195.24,Z 425.847,A -85,B 0,C 180,E1 -21957.938,E2 -21957.938} C_VEL
LIN {X 0,Y 195.301,Z 425.244,A -85,B 0,C 180,E1 -21960.001,E2 -21960.001} C_VEL
LIN {X 0,Y 194.82,Z 424.479,A -85,B 0,C 180,E1 -21964.138,E2 -21964.138} C_VEL
LIN {X 0,Y 194.718,Z 423.974,A -85,B 0,C 180,E1 -21968.302,E2 -21968.302} C_VEL
LIN {X 0,Y 194.478,Z 423.926,A -85,B 0,C 180,E1 -21972.679,E2 -21972.679} C_VEL
LIN {X 0,Y 194.497,Z 424.229,A -85,B 0,C 180,E1 -21976.803,E2 -21976.803} C_VEL
LIN {X 0,Y 194.603,Z 424.98,A -85,B 0,C 180,E1 -21981.171,E2 -21981.171} C_VEL
LIN {X 0,Y 194.839,Z 426.212,A -85,B 0,C 180,E1 -21985.649,E2 -21985.649} C_VEL
LIN {X 0,Y 195.164,Z 428,A -85,B 0,C 180,E1 -21990.276,E2 -21990.276} C_VEL
LIN {X 0,Y 195.613,Z 430.408,A -85,B 0,C 180,E1 -21995.09,E2 -21995.09} C_VEL
LIN {X 0,Y 195.918,Z 432.064,A -85,B 0,C 180,E1 -21997.9,E2 -21997.9} C_VEL
LIN {X 0,Y 196.568,Z 435.426,A -85,B 0,C 180,E1 -22002.791,E2 -22002.791} C_VEL
LIN {X 0,Y 197.209,Z 438.571,A -85,B 0,C 180,E1 -22006.779,E2 -22006.779} C_VEL
LIN {X 0,Y 198.752,Z 442.093,A -85,B 0,C 180,E1 -22007.63,E2 -22007.63} C_VEL
LIN {X 0,Y 200.584,Z 444.749,A -85,B 0,C 180,E1 -22008.488,E2 -22008.488} C_VEL
LIN {X 0,Y 202.844,Z 449.07,A -85,B 0,C 180,E1 -22009.663,E2 -22009.663} C_VEL
LIN {X 0,Y 205.867,Z 455.7,A -85,B 0,C 180,E1 -22011.346,E2 -22011.346} C_VEL
LIN {X 0,Y 207.212,Z 458.828,A -85,B 0,C 180,E1 -22012.131,E2 -22012.131} C_VEL
LIN {X 0,Y 208.444,Z 466.367,A -85,B 0,C 180,E1 -22013.554,E2 -22013.554} C_VEL
LIN {X 0,Y 209.033,Z 476.453,A -85,B 0,C 180,E1 -22015.482,E2 -22015.482} C_VEL
LIN {X 0,Y 208.608,Z 487.243,A -85,B 0,C 180,E1 -22017.705,E2 -22017.705} C_VEL
LIN {X 0,Y 207.179,Z 497.171,A -85,B 0,C 180,E1 -22019.982,E2 -22019.982} C_VEL
LIN {X 0,Y 206.05,Z 501.072,A -85,B 0,C 180,E1 -22020.925,E2 -22020.925} C_VEL
LIN {X 0,Y 202.69,Z 509.597,A -85,B 0,C 180,E1 -22023.213,E2 -22023.213} C_VEL
LIN {X 0,Y 199.191,Z 517.813,A -85,B 0,C 180,E1 -22026.067,E2 -22026.067} C_VEL
LIN {X 0,Y 196.494,Z 524.408,A -85,B 0,C 180,E1 -22029.048,E2 -22029.048} C_VEL
LIN {X 0,Y 195.789,Z 525.9,A -85,B 0,C 180,E1 -22029.843,E2 -22029.843} C_VEL
LIN {X 0,Y 193.939,Z 528.543,A -85,B 0,C 180,E1 -22031.303,E2 -22031.303} C_VEL
LIN {X 0,Y 189.456,Z 532.231,A -85,B 0,C 180,E1 -22033.712,E2 -22033.712} C_VEL
LIN {X 0,Y 185.341,Z 535.162,A -85,B 0,C 180,E1 -22036.32,E2 -22036.32} C_VEL
LIN {X 0,Y 184.105,Z 536.518,A -85,B 0,C 180,E1 -22038.053,E2 -22038.053} C_VEL
LIN {X 0,Y 183.474,Z 538.381,A -85,B 0,C 180,E1 -22041.192,E2 -22041.192} C_VEL
LIN {X 0,Y 183.303,Z 539.407,A -85,B 0,C 180,E1 -22044.229,E2 -22044.229} C_VEL
LIN {X 0,Y 183.272,Z 543.184,A -85,B 0,C 180,E1 -22047.807,E2 -22047.807} C_VEL
LIN {X 0,Y 183.415,Z 544.884,A -85,B 0,C 180,E1 -22050.005,E2 -22050.005} C_VEL
LIN {X 0,Y 183.114,Z 546.736,A -85,B 0,C 180,E1 -22053.71,E2 -22053.71} C_VEL
LIN {X 0,Y 183.218,Z 547.418,A -85,B 0,C 180,E1 -22056.613,E2 -22056.613} C_VEL
LIN {X 0,Y 184.092,Z 547.15,A -85,B 0,C 180,E1 -22061.009,E2 -22061.009} C_VEL
LIN {X 0,Y 185.9,Z 545.394,A -85,B 0,C 180,E1 -22065.35,E2 -22065.35} C_VEL
LIN {X 0,Y 187.211,Z 543.959,A -85,B 0,C 180,E1 -22067.482,E2 -22067.482} C_VEL
LIN {X 0,Y 190.858,Z 539.856,A -85,B 0,C 180,E1 -22071.611,E2 -22071.611} C_VEL
LIN {X 0,Y 194.169,Z 535.681,A -85,B 0,C 180,E1 -22074.602,E2 -22074.602} C_VEL
LIN {X 0,Y 197.872,Z 530.461,A -85,B 0,C 180,E1 -22077.503,E2 -22077.503} C_VEL
LIN {X 0,Y 202.349,Z 524.084,A -85,B 0,C 180,E1 -22080.244,E2 -22080.244} C_VEL
LIN {X 0,Y 207.312,Z 516.333,A -85,B 0,C 180,E1 -22082.852,E2 -22082.852} C_VEL
LIN {X 0,Y 211.903,Z 508.534,A -85,B 0,C 180,E1 -22084.902,E2 -22084.902} C_VEL
LIN {X 0,Y 215.446,Z 499.314,A -85,B 0,C 180,E1 -22087.338,E2 -22087.338} C_VEL
LIN {X 0,Y 218.356,Z 488.251,A -85,B 0,C 180,E1 -22090.074,E2 -22090.074} C_VEL
LIN {X 0,Y 219.072,Z 483.356,A -85,B 0,C 180,E1 -22091.371,E2 -22091.371} C_VEL
LIN {X 0,Y 218.832,Z 480.625,A -85,B 0,C 180,E1 -22092.381,E2 -22092.381} C_VEL
LIN {X 0,Y 217.308,Z 473.961,A -85,B 0,C 180,E1 -22095.362,E2 -22095.362} C_VEL
LIN {X 0,Y 216.074,Z 469.83,A -85,B 0,C 180,E1 -22097.586,E2 -22097.586} C_VEL
LIN {X 0,Y 215.183,Z 467.377,A -85,B 0,C 180,E1 -22099.215,E2 -22099.215} C_VEL
LIN {X 0,Y 213.907,Z 465.027,A -85,B 0,C 180,E1 -22101.372,E2 -22101.372} C_VEL
LIN {X 0,Y 212.114,Z 461.46,A -85,B 0,C 180,E1 -22105.933,E2 -22105.933} C_VEL
LIN {X 0,Y 211.606,Z 460.673,A -85,B 0,C 180,E1 -22107.899,E2 -22107.899} C_VEL
LIN {X 0,Y 211.375,Z 460.354,A -85,B 0,C 180,E1 -22112.258,E2 -22112.258} C_VEL
LIN {X 0,Y 211.478,Z 461.223,A -85,B 0,C 180,E1 -22114.403,E2 -22114.403} C_VEL
LIN {X 0,Y 212.597,Z 463.924,A -85,B 0,C 180,E1 -22118.676,E2 -22118.676} C_VEL
LIN {X 0,Y 213.492,Z 465.902,A -85,B 0,C 180,E1 -22120.78,E2 -22120.78} C_VEL
LIN {X 0,Y 214.982,Z 470.049,A -85,B 0,C 180,E1 -22123.967,E2 -22123.967} C_VEL
LIN {X 0,Y 216.47,Z 474.954,A -85,B 0,C 180,E1 -22126.916,E2 -22126.916} C_VEL
LIN {X 0,Y 216.947,Z 476.885,A -85,B 0,C 180,E1 -22127.921,E2 -22127.921} C_VEL
LIN {X 0,Y 217.19,Z 481.256,A -85,B 0,C 180,E1 -22129.688,E2 -22129.688} C_VEL
LIN {X 0,Y 216.354,Z 491.346,A -85,B 0,C 180,E1 -22133.206,E2 -22133.206} C_VEL
LIN {X 0,Y 215.274,Z 497.643,A -85,B 0,C 180,E1 -22135.318,E2 -22135.318} C_VEL
LIN {X 0,Y 214.916,Z 499.016,A -85,B 0,C 180,E1 -22135.78,E2 -22135.78} C_VEL
LIN {X 0,Y 211.028,Z 506.181,A -85,B 0,C 180,E1 -22137.646,E2 -22137.646} C_VEL
LIN {X 0,Y 206.264,Z 513.746,A -85,B 0,C 180,E1 -22139.999,E2 -22139.999} C_VEL
LIN {X 0,Y 201.029,Z 521.261,A -85,B 0,C 180,E1 -22143.005,E2 -22143.005} C_VEL
LIN {X 0,Y 196.526,Z 527.143,A -85,B 0,C 180,E1 -22146.158,E2 -22146.158} C_VEL
LIN {X 0,Y 192.47,Z 531.859,A -85,B 0,C 180,E1 -22149.614,E2 -22149.614} C_VEL
LIN {X 0,Y 189.403,Z 535.019,A -85,B 0,C 180,E1 -22152.863,E2 -22152.863} C_VEL
LIN {X 0,Y 187.614,Z 536.632,A -85,B 0,C 180,E1 -22155.201,E2 -22155.201} C_VEL
LIN {X 0,Y 185.521,Z 538.116,A -85,B 0,C 180,E1 -22158.716,E2 -22158.716} C_VEL
LIN {X 0,Y 183.736,Z 538.497,A -85,B 0,C 180,E1 -22163.354,E2 -22163.354} C_VEL
LIN {X 0,Y 182.842,Z 537.254,A -85,B 0,C 180,E1 -22167.856,E2 -22167.856} C_VEL
LIN {X 0,Y 182.643,Z 534.482,A -85,B 0,C 180,E1 -22172.155,E2 -22172.155} C_VEL
LIN {X 0,Y 183.092,Z 530.349,A -85,B 0,C 180,E1 -22176.279,E2 -22176.279} C_VEL
LIN {X 0,Y 183.841,Z 524.886,A -85,B 0,C 180,E1 -22180.125,E2 -22180.125} C_VEL
LIN {X 0,Y 184.848,Z 518.178,A -85,B 0,C 180,E1 -22183.742,E2 -22183.742} C_VEL
LIN {X 0,Y 186.031,Z 511.522,A -85,B 0,C 180,E1 -22186.613,E2 -22186.613} C_VEL
LIN {X 0,Y 187.725,Z 502.637,A -85,B 0,C 180,E1 -22189.71,E2 -22189.71} C_VEL
LIN {X 0,Y 189.623,Z 493.054,A -85,B 0,C 180,E1 -22192.392,E2 -22192.392} C_VEL
LIN {X 0,Y 191.596,Z 482.512,A -85,B 0,C 180,E1 -22194.778,E2 -22194.778} C_VEL
LIN {X 0,Y 192.643,Z 476.679,A -85,B 0,C 180,E1 -22195.876,E2 -22195.876} C_VEL
LIN {X 0,Y 192.087,Z 468.908,A -85,B 0,C 180,E1 -22197.299,E2 -22197.299} C_VEL
LIN {X 0,Y 190.595,Z 457.184,A -85,B 0,C 180,E1 -22199.149,E2 -22199.149} C_VEL
LIN {X 0,Y 188.529,Z 443.813,A -85,B 0,C 180,E1 -22200.861,E2 -22200.861} C_VEL
LIN {X 0,Y 186.04,Z 430.585,A -85,B 0,C 180,E1 -22202.2,E2 -22202.2} C_VEL
LIN {X 0,Y 186.704,Z 424.959,A -85,B 0,C 180,E1 -22206.714,E2 -22206.714} C_VEL
LIN {X 0,Y 186.624,Z 422.164,A -85,B 0,C 180,E1 -22209.033,E2 -22209.033} C_VEL
LIN {X 0,Y 185.772,Z 417.344,A -85,B 0,C 180,E1 -22213.229,E2 -22213.229} C_VEL
LIN {X 0,Y 185.824,Z 417.443,A -85,B 0,C 180,E1 -22217.989,E2 -22217.989} C_VEL
LIN {X 0,Y 186.351,Z 419.865,A -85,B 0,C 180,E1 -22221.319,E2 -22221.319} C_VEL
LIN {X 0,Y 186.909,Z 423.204,A -85,B 0,C 180,E1 -22225.682,E2 -22225.682} C_VEL
LIN {X 0,Y 187.272,Z 424.921,A -85,B 0,C 180,E1 -22227.845,E2 -22227.845} C_VEL
LIN {X 0,Y 186.387,Z 428.729,A -85,B 0,C 180,E1 -22232.156,E2 -22232.156} C_VEL
LIN {X 0,Y 186.145,Z 430.038,A -85,B 0,C 180,E1 -22233.445,E2 -22233.445} C_VEL
LIN {X 0,Y 188.945,Z 441.236,A -85,B 0,C 180,E1 -22234.796,E2 -22234.796} C_VEL
LIN {X 0,Y 190.929,Z 452.017,A -85,B 0,C 180,E1 -22236.362,E2 -22236.362} C_VEL
LIN {X 0,Y 192.419,Z 463.485,A -85,B 0,C 180,E1 -22238.396,E2 -22238.396} C_VEL
LIN {X 0,Y 193.051,Z 471.193,A -85,B 0,C 180,E1 -22240.006,E2 -22240.006} C_VEL
LIN {X 0,Y 191.151,Z 481.011,A -85,B 0,C 180,E1 -22242.2,E2 -22242.2} C_VEL
LIN {X 0,Y 189.083,Z 490.416,A -85,B 0,C 180,E1 -22244.9,E2 -22244.9} C_VEL
LIN {X 0,Y 187.476,Z 497.448,A -85,B 0,C 180,E1 -22247.446,E2 -22247.446} C_VEL
LIN {X 0,Y 185.927,Z 504.015,A -85,B 0,C 180,E1 -22250.46,E2 -22250.46} C_VEL
LIN {X 0,Y 184.883,Z 508.638,A -85,B 0,C 180,E1 -22253.141,E2 -22253.141} C_VEL
LIN {X 0,Y 184.05,Z 512.548,A -85,B 0,C 180,E1 -22256.042,E2 -22256.042} C_VEL
LIN {X 0,Y 183.394,Z 516.213,A -85,B 0,C 180,E1 -22259.873,E2 -22259.873} C_VEL
LIN {X 0,Y 183.256,Z 517.832,A -85,B 0,C 180,E1 -22262.467,E2 -22262.467} C_VEL
LIN {X 0,Y 183.572,Z 519.002,A -85,B 0,C 180,E1 -22266.489,E2 -22266.489} C_VEL
LIN {X 0,Y 184.52,Z 518.692,A -85,B 0,C 180,E1 -22270.382,E2 -22270.382} C_VEL
LIN {X 0,Y 186.038,Z 516.962,A -85,B 0,C 180,E1 -22274.131,E2 -22274.131} C_VEL
LIN {X 0,Y 188.121,Z 513.895,A -85,B 0,C 180,E1 -22277.744,E2 -22277.744} C_VEL
LIN {X 0,Y 190.719,Z 509.403,A -85,B 0,C 180,E1 -22281.212,E2 -22281.212} C_VEL
LIN {X 0,Y 193.281,Z 504.601,A -85,B 0,C 180,E1 -22283.944,E2 -22283.944} C_VEL
LIN {X 0,Y 196.863,Z 497.389,A -85,B 0,C 180,E1 -22287.019,E2 -22287.019} C_VEL
LIN {X 0,Y 200.454,Z 489.202,A -85,B 0,C 180,E1 -22289.685,E2 -22289.685} C_VEL
LIN {X 0,Y 202.183,Z 484.723,A -85,B 0,C 180,E1 -22290.88,E2 -22290.88} C_VEL
LIN {X 0,Y 202.797,Z 478.672,A -85,B 0,C 180,E1 -22292.666,E2 -22292.666} C_VEL
LIN {X 0,Y 202.452,Z 470.167,A -85,B 0,C 180,E1 -22295.081,E2 -22295.081} C_VEL
LIN {X 0,Y 200.957,Z 460.606,A -85,B 0,C 180,E1 -22297.724,E2 -22297.724} C_VEL
LIN {X 0,Y 198.818,Z 452.701,A -85,B 0,C 180,E1 -22299.937,E2 -22299.937} C_VEL
LIN {X 0,Y 195.786,Z 445.282,A -85,B 0,C 180,E1 -22302.235,E2 -22302.235} C_VEL
LIN {X 0,Y 194.413,Z 442.309,A -85,B 0,C 180,E1 -22303.191,E2 -22303.191} C_VEL
LIN {X 0,Y 192.293,Z 438.797,A -85,B 0,C 180,E1 -22304.499,E2 -22304.499} C_VEL
LIN {X 0,Y 191.464,Z 437.259,A -85,B 0,C 180,E1 -22305.044,E2 -22305.044} C_VEL
LIN {X 0,Y 189.308,Z 434.262,A -85,B 0,C 180,E1 -22306.335,E2 -22306.335} C_VEL
LIN {X 0,Y 188.606,Z 432.273,A -85,B 0,C 180,E1 -22306.975,E2 -22306.975} C_VEL
LIN {X 0,Y 188.53,Z 430.282,A -85,B 0,C 180,E1 -22311.425,E2 -22311.425} C_VEL
LIN {X 0,Y 188.401,Z 428.684,A -85,B 0,C 180,E1 -22315.722,E2 -22315.722} C_VEL
LIN {X 0,Y 188.523,Z 427.387,A -85,B 0,C 180,E1 -22320.001,E2 -22320.001} C_VEL
LIN {X 0,Y 188.055,Z 426.66,A -85,B 0,C 180,E1 -22324.287,E2 -22324.287} C_VEL
LIN {X 0,Y 187.966,Z 426.204,A -85,B 0,C 180,E1 -22328.602,E2 -22328.602} C_VEL
LIN {X 0,Y 187.745,Z 426.226,A -85,B 0,C 180,E1 -22333.303,E2 -22333.303} C_VEL
LIN {X 0,Y 187.77,Z 426.596,A -85,B 0,C 180,E1 -22337.424,E2 -22337.424} C_VEL
LIN {X 0,Y 187.885,Z 427.446,A -85,B 0,C 180,E1 -22341.967,E2 -22341.967} C_VEL
LIN {X 0,Y 188.108,Z 428.81,A -85,B 0,C 180,E1 -22346.638,E2 -22346.638} C_VEL
LIN {X 0,Y 188.469,Z 430.742,A -85,B 0,C 180,E1 -22351.471,E2 -22351.471} C_VEL
LIN {X 0,Y 188.846,Z 432.513,A -85,B 0,C 180,E1 -22355.052,E2 -22355.052} C_VEL
LIN {X 0,Y 189.265,Z 434.946,A -85,B 0,C 180,E1 -22359.144,E2 -22359.144} C_VEL
LIN {X 0,Y 189.991,Z 438.297,A -85,B 0,C 180,E1 -22363.918,E2 -22363.918} C_VEL
LIN {X 0,Y 191.515,Z 441.645,A -85,B 0,C 180,E1 -22364.877,E2 -22364.877} C_VEL
LIN {X 0,Y 193.596,Z 444.447,A -85,B 0,C 180,E1 -22365.987,E2 -22365.987} C_VEL
LIN {X 0,Y 195.537,Z 448.375,A -85,B 0,C 180,E1 -22367.175,E2 -22367.175} C_VEL
LIN {X 0,Y 196.706,Z 450.524,A -85,B 0,C 180,E1 -22367.842,E2 -22367.842} C_VEL
LIN {X 0,Y 200.767,Z 459.305,A -85,B 0,C 180,E1 -22370.366,E2 -22370.366} C_VEL
LIN {X 0,Y 202.233,Z 463.36,A -85,B 0,C 180,E1 -22371.436,E2 -22371.436} C_VEL
LIN {X 0,Y 203.124,Z 472.929,A -85,B 0,C 180,E1 -22373.369,E2 -22373.369} C_VEL
LIN {X 0,Y 203.021,Z 483.001,A -85,B 0,C 180,E1 -22375.483,E2 -22375.483} C_VEL
LIN {X 0,Y 201.96,Z 492.654,A -85,B 0,C 180,E1 -22377.692,E2 -22377.692} C_VEL
LIN {X 0,Y 200.58,Z 499.65,A -85,B 0,C 180,E1 -22379.472,E2 -22379.472} C_VEL
LIN {X 0,Y 197.084,Z 508.354,A -85,B 0,C 180,E1 -22381.81,E2 -22381.81} C_VEL
LIN {X 0,Y 193.846,Z 515.51,A -85,B 0,C 180,E1 -22384.216,E2 -22384.216} C_VEL
LIN {X 0,Y 190.941,Z 521.905,A -85,B 0,C 180,E1 -22386.954,E2 -22386.954} C_VEL
LIN {X 0,Y 188.943,Z 526.302,A -85,B 0,C 180,E1 -22389.312,E2 -22389.312} C_VEL
LIN {X 0,Y 186.675,Z 531.029,A -85,B 0,C 180,E1 -22392.477,E2 -22392.477} C_VEL
LIN {X 0,Y 184.891,Z 534.629,A -85,B 0,C 180,E1 -22395.701,E2 -22395.701} C_VEL
LIN {X 0,Y 184.105,Z 536.518,A -85,B 0,C 180,E1 -22398.053,E2 -22398.053} C_VEL
LIN {X 0,Y 183.028,Z 537.695,A -85,B 0,C 180,E1 -22399.825,E2 -22399.825} C_VEL
LIN {X 0,Y 179.777,Z 539.167,A -85,B 0,C 180,E1 -22402.74,E2 -22402.74} C_VEL
LIN {X 0,Y 177.259,Z 540.477,A -85,B 0,C 180,E1 -22405.126,E2 -22405.126} C_VEL
LIN {X 0,Y 176.248,Z 541.831,A -85,B 0,C 180,E1 -22406.967,E2 -22406.967} C_VEL
LIN {X 0,Y 176.19,Z 542.375,A -85,B 0,C 180,E1 -22407.582,E2 -22407.582} C_VEL
LIN {X 0,Y 176.352,Z 544.325,A -85,B 0,C 180,E1 -22410.005,E2 -22410.005} C_VEL
LIN {X 0,Y 176.054,Z 546.232,A -85,B 0,C 180,E1 -22413.623,E2 -22413.623} C_VEL
LIN {X 0,Y 176.147,Z 547.098,A -85,B 0,C 180,E1 -22416.879,E2 -22416.879} C_VEL
LIN {X 0,Y 177.094,Z 547.065,A -85,B 0,C 180,E1 -22421.45,E2 -22421.45} C_VEL
LIN {X 0,Y 179.034,Z 545.491,A -85,B 0,C 180,E1 -22425.954,E2 -22425.954} C_VEL
LIN {X 0,Y 182.236,Z 542.452,A -85,B 0,C 180,E1 -22430.314,E2 -22430.314} C_VEL
LIN {X 0,Y 185.414,Z 539.093,A -85,B 0,C 180,E1 -22433.458,E2 -22433.458} C_VEL
LIN {X 0,Y 189.396,Z 534.303,A -85,B 0,C 180,E1 -22436.841,E2 -22436.841} C_VEL
LIN {X 0,Y 193.875,Z 528.516,A -85,B 0,C 180,E1 -22439.901,E2 -22439.901} C_VEL
LIN {X 0,Y 199.701,Z 520.45,A -85,B 0,C 180,E1 -22443.062,E2 -22443.062} C_VEL
LIN {X 0,Y 205.349,Z 512.008,A -85,B 0,C 180,E1 -22445.583,E2 -22445.583} C_VEL
LIN {X 0,Y 207.795,Z 507.283,A -85,B 0,C 180,E1 -22446.898,E2 -22446.898} C_VEL
LIN {X 0,Y 211.151,Z 498.704,A -85,B 0,C 180,E1 -22449.232,E2 -22449.232} C_VEL
LIN {X 0,Y 213.878,Z 489.451,A -85,B 0,C 180,E1 -22451.663,E2 -22451.663} C_VEL
LIN {X 0,Y 214.279,Z 486.039,A -85,B 0,C 180,E1 -22452.743,E2 -22452.743} C_VEL
LIN {X 0,Y 213.068,Z 478.906,A -85,B 0,C 180,E1 -22456.156,E2 -22456.156} C_VEL
LIN {X 0,Y 212.112,Z 474.951,A -85,B 0,C 180,E1 -22458.495,E2 -22458.495} C_VEL
LIN {X 0,Y 211.048,Z 472.012,A -85,B 0,C 180,E1 -22460.749,E2 -22460.749} C_VEL
LIN {X 0,Y 209.307,Z 468.484,A -85,B 0,C 180,E1 -22465.192,E2 -22465.192} C_VEL
LIN {X 0,Y 208.805,Z 467.34,A -85,B 0,C 180,E1 -22467.415,E2 -22467.415} C_VEL
LIN {X 0,Y 208.431,Z 466.8,A -85,B 0,C 180,E1 -22471.831,E2 -22471.831} C_VEL
LIN {X 0,Y 208.495,Z 467.518,A -85,B 0,C 180,E1 -22474.01,E2 -22474.01} C_VEL
LIN {X 0,Y 209.26,Z 470.067,A -85,B 0,C 180,E1 -22478.319,E2 -22478.319} C_VEL
LIN {X 0,Y 210.01,Z 471.965,A -85,B 0,C 180,E1 -22480.448,E2 -22480.448} C_VEL
LIN {X 0,Y 211.129,Z 475.963,A -85,B 0,C 180,E1 -22483.666,E2 -22483.666} C_VEL
LIN {X 0,Y 212.198,Z 480.577,A -85,B 0,C 180,E1 -22486.594,E2 -22486.594} C_VEL
LIN {X 0,Y 212.49,Z 483.599,A -85,B 0,C 180,E1 -22488.109,E2 -22488.109} C_VEL
LIN {X 0,Y 211.844,Z 489.764,A -85,B 0,C 180,E1 -22490.451,E2 -22490.451} C_VEL
LIN {X 0,Y 210.562,Z 497.355,A -85,B 0,C 180,E1 -22493.291,E2 -22493.291} C_VEL
LIN {X 0,Y 209.462,Z 501.338,A -85,B 0,C 180,E1 -22494.705,E2 -22494.705} C_VEL
LIN {X 0,Y 204.07,Z 510.184,A -85,B 0,C 180,E1 -22497.18,E2 -22497.18} C_VEL
LIN {X 0,Y 198.469,Z 518.072,A -85,B 0,C 180,E1 -22499.999,E2 -22499.999} C_VEL
LIN {X 0,Y 193.223,Z 524.722,A -85,B 0,C 180,E1 -22503.127,E2 -22503.127} C_VEL
LIN {X 0,Y 188.701,Z 529.879,A -85,B 0,C 180,E1 -22506.414,E2 -22506.414} C_VEL
LIN {X 0,Y 185.256,Z 533.398,A -85,B 0,C 180,E1 -22509.456,E2 -22509.456} C_VEL
LIN {X 0,Y 181.706,Z 536.505,A -85,B 0,C 180,E1 -22513.418,E2 -22513.418} C_VEL
LIN {X 0,Y 179.959,Z 537.758,A -85,B 0,C 180,E1 -22515.864,E2 -22515.864} C_VEL
LIN {X 0,Y 178.273,Z 538.597,A -85,B 0,C 180,E1 -22518.878,E2 -22518.878} C_VEL
LIN {X 0,Y 176.597,Z 538.608,A -85,B 0,C 180,E1 -22523.45,E2 -22523.45} C_VEL
LIN {X 0,Y 175.974,Z 537.891,A -85,B 0,C 180,E1 -22526.059,E2 -22526.059} C_VEL
LIN {X 0,Y 175.644,Z 536.69,A -85,B 0,C 180,E1 -22528.695,E2 -22528.695} C_VEL
LIN {X 0,Y 175.574,Z 533.749,A -85,B 0,C 180,E1 -22532.789,E2 -22532.789} C_VEL
LIN {X 0,Y 176.094,Z 529.2,A -85,B 0,C 180,E1 -22537.034,E2 -22537.034} C_VEL
LIN {X 0,Y 176.916,Z 523.446,A -85,B 0,C 180,E1 -22540.988,E2 -22540.988} C_VEL
LIN {X 0,Y 178.087,Z 516.308,A -85,B 0,C 180,E1 -22544.731,E2 -22544.731} C_VEL
LIN {X 0,Y 179.736,Z 507.571,A -85,B 0,C 180,E1 -22548.333,E2 -22548.333} C_VEL
LIN {X 0,Y 181.577,Z 498.323,A -85,B 0,C 180,E1 -22551.335,E2 -22551.335} C_VEL
LIN {X 0,Y 183.618,Z 488.083,A -85,B 0,C 180,E1 -22554.014,E2 -22554.014} C_VEL
LIN {X 0,Y 185.718,Z 476.797,A -85,B 0,C 180,E1 -22556.358,E2 -22556.358} C_VEL
LIN {X 0,Y 184.851,Z 467.263,A -85,B 0,C 180,E1 -22558.157,E2 -22558.157} C_VEL
LIN {X 0,Y 183.286,Z 455.095,A -85,B 0,C 180,E1 -22560.096,E2 -22560.096} C_VEL
LIN {X 0,Y 181.217,Z 441.937,A -85,B 0,C 180,E1 -22561.788,E2 -22561.788} C_VEL
LIN {X 0,Y 179.112,Z 430.702,A -85,B 0,C 180,E1 -22562.951,E2 -22562.951} C_VEL
LIN {X 0,Y 179.705,Z 425.808,A -85,B 0,C 180,E1 -22566.973,E2 -22566.973} C_VEL
LIN {X 0,Y 179.562,Z 423.025,A -85,B 0,C 180,E1 -22569.37,E2 -22569.37} C_VEL
LIN {X 0,Y 178.716,Z 418.224,A -85,B 0,C 180,E1 -22573.724,E2 -22573.724} C_VEL
LIN {X 0,Y 178.739,Z 418.371,A -85,B 0,C 180,E1 -22577.217,E2 -22577.217} C_VEL
LIN {X 0,Y 179.315,Z 420.974,A -85,B 0,C 180,E1 -22580.975,E2 -22580.975} C_VEL
LIN {X 0,Y 179.899,Z 424.349,A -85,B 0,C 180,E1 -22585.514,E2 -22585.514} C_VEL
LIN {X 0,Y 180.259,Z 426.061,A -85,B 0,C 180,E1 -22587.761,E2 -22587.761} C_VEL
LIN {X 0,Y 179.277,Z 430.067,A -85,B 0,C 180,E1 -22592.452,E2 -22592.452} C_VEL
LIN {X 0,Y 182.483,Z 443.174,A -85,B 0,C 180,E1 -22594.136,E2 -22594.136} C_VEL
LIN {X 0,Y 184.444,Z 454.747,A -85,B 0,C 180,E1 -22595.955,E2 -22595.955} C_VEL
LIN {X 0,Y 185.695,Z 464.936,A -85,B 0,C 180,E1 -22597.88,E2 -22597.88} C_VEL
LIN {X 0,Y 186.185,Z 471.669,A -85,B 0,C 180,E1 -22599.364,E2 -22599.364} C_VEL
LIN {X 0,Y 184.924,Z 478.676,A -85,B 0,C 180,E1 -22600.949,E2 -22600.949} C_VEL
LIN {X 0,Y 182.985,Z 487.356,A -85,B 0,C 180,E1 -22603.318,E2 -22603.318} C_VEL
LIN {X 0,Y 180.935,Z 496.056,A -85,B 0,C 180,E1 -22606.351,E2 -22606.351} C_VEL
LIN {X 0,Y 179.505,Z 501.95,A -85,B 0,C 180,E1 -22608.941,E2 -22608.941} C_VEL
LIN {X 0,Y 178.126,Z 507.537,A -85,B 0,C 180,E1 -22612.007,E2 -22612.007} C_VEL
LIN {X 0,Y 176.995,Z 512.806,A -85,B 0,C 180,E1 -22615.892,E2 -22615.892} C_VEL
LIN {X 0,Y 176.43,Z 515.665,A -85,B 0,C 180,E1 -22618.796,E2 -22618.796} C_VEL
LIN {X 0,Y 176.184,Z 517.442,A -85,B 0,C 180,E1 -22621.23,E2 -22621.23} C_VEL
LIN {X 0,Y 176.211,Z 518.736,A -85,B 0,C 180,E1 -22623.936,E2 -22623.936} C_VEL
LIN {X 0,Y 176.645,Z 519.462,A -85,B 0,C 180,E1 -22627.278,E2 -22627.278} C_VEL
LIN {X 0,Y 177.702,Z 519.014,A -85,B 0,C 180,E1 -22631.286,E2 -22631.286} C_VEL
LIN {X 0,Y 179.419,Z 517.198,A -85,B 0,C 180,E1 -22635.165,E2 -22635.165} C_VEL
LIN {X 0,Y 181.677,Z 514.015,A -85,B 0,C 180,E1 -22638.882,E2 -22638.882} C_VEL
LIN {X 0,Y 184.555,Z 509.432,A -85,B 0,C 180,E1 -22642.463,E2 -22642.463} C_VEL
LIN {X 0,Y 187.98,Z 503.251,A -85,B 0,C 180,E1 -22645.889,E2 -22645.889} C_VEL
LIN {X 0,Y 191.437,Z 496.671,A -85,B 0,C 180,E1 -22648.608,E2 -22648.608} C_VEL
LIN {X 0,Y 195.282,Z 488.207,A -85,B 0,C 180,E1 -22651.291,E2 -22651.291} C_VEL
LIN {X 0,Y 196.305,Z 484.872,A -85,B 0,C 180,E1 -22652.263,E2 -22652.263} C_VEL
LIN {X 0,Y 196.822,Z 478.537,A -85,B 0,C 180,E1 -22654.236,E2 -22654.236} C_VEL
LIN {X 0,Y 196.37,Z 470.106,A -85,B 0,C 180,E1 -22656.817,E2 -22656.817} C_VEL
LIN {X 0,Y 195.062,Z 461.466,A -85,B 0,C 180,E1 -22659.366,E2 -22659.366} C_VEL
LIN {X 0,Y 192.972,Z 454.035,A -85,B 0,C 180,E1 -22661.693,E2 -22661.693} C_VEL
LIN {X 0,Y 189.844,Z 446.912,A -85,B 0,C 180,E1 -22664.24,E2 -22664.24} C_VEL
LIN {X 0,Y 187.615,Z 442.707,A -85,B 0,C 180,E1 -22665.902,E2 -22665.902} C_VEL
LIN {X 0,Y 185.538,Z 439.133,A -85,B 0,C 180,E1 -22667.421,E2 -22667.421} C_VEL
LIN {X 0,Y 184.873,Z 437.914,A -85,B 0,C 180,E1 -22667.932,E2 -22667.932} C_VEL
LIN {X 0,Y 182.712,Z 435.166,A -85,B 0,C 180,E1 -22669.403,E2 -22669.403} C_VEL
LIN {X 0,Y 181.715,Z 432.729,A -85,B 0,C 180,E1 -22670.4,E2 -22670.4} C_VEL
LIN {X 0,Y 181.613,Z 430.855,A -85,B 0,C 180,E1 -22675.562,E2 -22675.562} C_VEL
LIN {X 0,Y 181.759,Z 429.541,A -85,B 0,C 180,E1 -22680.001,E2 -22680.001} C_VEL
LIN {X 0,Y 181.304,Z 428.835,A -85,B 0,C 180,E1 -22684.447,E2 -22684.447} C_VEL
LIN {X 0,Y 181.195,Z 428.439,A -85,B 0,C 180,E1 -22688.926,E2 -22688.926} C_VEL
LIN {X 0,Y 180.999,Z 428.533,A -85,B 0,C 180,E1 -22693.924,E2 -22693.924} C_VEL
LIN {X 0,Y 181.051,Z 428.969,A -85,B 0,C 180,E1 -22698.093,E2 -22698.093} C_VEL
LIN {X 0,Y 181.159,Z 429.577,A -85,B 0,C 180,E1 -22701.415,E2 -22701.415} C_VEL
LIN {X 0,Y 181.305,Z 430.586,A -85,B 0,C 180,E1 -22705.24,E2 -22705.24} C_VEL
LIN {X 0,Y 181.609,Z 432.382,A -85,B 0,C 180,E1 -22710.205,E2 -22710.205} C_VEL
LIN {X 0,Y 182.15,Z 435.101,A -85,B 0,C 180,E1 -22715.889,E2 -22715.889} C_VEL
LIN {X 0,Y 182.637,Z 437.979,A -85,B 0,C 180,E1 -22720.403,E2 -22720.403} C_VEL
LIN {X 0,Y 184.12,Z 441.151,A -85,B 0,C 180,E1 -22721.525,E2 -22721.525} C_VEL
LIN {X 0,Y 186.662,Z 444.352,A -85,B 0,C 180,E1 -22723.119,E2 -22723.119} C_VEL
LIN {X 0,Y 188.75,Z 448.369,A -85,B 0,C 180,E1 -22724.559,E2 -22724.559} C_VEL
LIN {X 0,Y 189.899,Z 450.268,A -85,B 0,C 180,E1 -22725.282,E2 -22725.282} C_VEL
LIN {X 0,Y 193.796,Z 458.576,A -85,B 0,C 180,E1 -22728.026,E2 -22728.026} C_VEL
LIN {X 0,Y 196.655,Z 465.879,A -85,B 0,C 180,E1 -22730.207,E2 -22730.207} C_VEL
LIN {X 0,Y 197.192,Z 468.595,A -85,B 0,C 180,E1 -22730.888,E2 -22730.888} C_VEL
LIN {X 0,Y 197.44,Z 478.668,A -85,B 0,C 180,E1 -22733.092,E2 -22733.092} C_VEL
LIN {X 0,Y 196.75,Z 488.049,A -85,B 0,C 180,E1 -22735.244,E2 -22735.244} C_VEL
LIN {X 0,Y 195.371,Z 496.397,A -85,B 0,C 180,E1 -22737.351,E2 -22737.351} C_VEL
LIN {X 0,Y 193.802,Z 502.073,A -85,B 0,C 180,E1 -22738.891,E2 -22738.891} C_VEL
LIN {X 0,Y 189.456,Z 511.684,A -85,B 0,C 180,E1 -22741.779,E2 -22741.779} C_VEL
LIN {X 0,Y 185.728,Z 519.318,A -85,B 0,C 180,E1 -22744.811,E2 -22744.811} C_VEL
LIN {X 0,Y 182.309,Z 526.332,A -85,B 0,C 180,E1 -22748.523,E2 -22748.523} C_VEL
LIN {X 0,Y 179.902,Z 530.959,A -85,B 0,C 180,E1 -22751.794,E2 -22751.794} C_VEL
LIN {X 0,Y 178.532,Z 533.389,A -85,B 0,C 180,E1 -22754.01,E2 -22754.01} C_VEL
LIN {X 0,Y 177.044,Z 536.489,A -85,B 0,C 180,E1 -22757.869,E2 -22757.869} C_VEL
LIN {X 0,Y 176.43,Z 538.062,A -85,B 0,C 180,E1 -22760.837,E2 -22760.837} C_VEL
LIN {X 0,Y 176.218,Z 539.265,A -85,B 0,C 180,E1 -22764.57,E2 -22764.57} C_VEL
LIN {X 0,Y 176.19,Z 542.375,A -85,B 0,C 180,E1 -22767.582,E2 -22767.582} C_VEL
LIN {X 0,Y 175.536,Z 543.916,A -85,B 0,C 180,E1 -22769.423,E2 -22769.423} C_VEL
LIN {X 0,Y 173.895,Z 545.064,A -85,B 0,C 180,E1 -22771.26,E2 -22771.26} C_VEL
LIN {X 0,Y 170.102,Z 546.416,A -85,B 0,C 180,E1 -22775.047,E2 -22775.047} C_VEL
LIN {X 0,Y 169.169,Z 546.764,A -85,B 0,C 180,E1 -22777.05,E2 -22777.05} C_VEL
LIN {X 0,Y 169.161,Z 546.837,A -85,B 0,C 180,E1 -22777.728,E2 -22777.728} C_VEL
LIN {X 0,Y 170.119,Z 546.916,A -85,B 0,C 180,E1 -22781.926,E2 -22781.926} C_VEL
LIN {X 0,Y 172.192,Z 545.598,A -85,B 0,C 180,E1 -22786.606,E2 -22786.606} C_VEL
LIN {X 0,Y 175.604,Z 542.744,A -85,B 0,C 180,E1 -22791.117,E2 -22791.117} C_VEL
LIN {X 0,Y 180.14,Z 538.391,A -85,B 0,C 180,E1 -22795.419,E2 -22795.419} C_VEL
LIN {X 0,Y 184.371,Z 533.615,A -85,B 0,C 180,E1 -22798.748,E2 -22798.748} C_VEL
LIN {X 0,Y 189.484,Z 527.509,A -85,B 0,C 180,E1 -22801.911,E2 -22801.911} C_VEL
LIN {X 0,Y 195.789,Z 519.373,A -85,B 0,C 180,E1 -22805.058,E2 -22805.058} C_VEL
LIN {X 0,Y 201.613,Z 510.763,A -85,B 0,C 180,E1 -22807.596,E2 -22807.596} C_VEL
LIN {X 0,Y 206.043,Z 501.15,A -85,B 0,C 180,E1 -22810.401,E2 -22810.401} C_VEL
LIN {X 0,Y 208.618,Z 494.051,A -85,B 0,C 180,E1 -22812.363,E2 -22812.363} C_VEL
LIN {X 0,Y 209.43,Z 490.378,A -85,B 0,C 180,E1 -22813.521,E2 -22813.521} C_VEL
LIN {X 0,Y 208.785,Z 484.384,A -85,B 0,C 180,E1 -22816.597,E2 -22816.597} C_VEL
LIN {X 0,Y 208.125,Z 480.44,A -85,B 0,C 180,E1 -22819.055,E2 -22819.055} C_VEL
LIN {X 0,Y 207.288,Z 477.833,A -85,B 0,C 180,E1 -22821.248,E2 -22821.248} C_VEL
LIN {X 0,Y 206.049,Z 474.988,A -85,B 0,C 180,E1 -22824.95,E2 -22824.95} C_VEL
LIN {X 0,Y 205.666,Z 473.97,A -85,B 0,C 180,E1 -22826.855,E2 -22826.855} C_VEL
LIN {X 0,Y 205.336,Z 473.312,A -85,B 0,C 180,E1 -22829.108,E2 -22829.108} C_VEL
LIN {X 0,Y 205.2,Z 473.114,A -85,B 0,C 180,E1 -22831.347,E2 -22831.347} C_VEL
LIN {X 0,Y 205.2,Z 473.685,A -85,B 0,C 180,E1 -22833.56,E2 -22833.56} C_VEL
LIN {X 0,Y 205.671,Z 476.064,A -85,B 0,C 180,E1 -22837.921,E2 -22837.921} C_VEL
LIN {X 0,Y 206.242,Z 477.815,A -85,B 0,C 180,E1 -22840.076,E2 -22840.076} C_VEL
LIN {X 0,Y 206.966,Z 481.355,A -85,B 0,C 180,E1 -22843.127,E2 -22843.127} C_VEL
LIN {X 0,Y 207.69,Z 486.065,A -85,B 0,C 180,E1 -22846.297,E2 -22846.297} C_VEL
LIN {X 0,Y 207.672,Z 488.674,A -85,B 0,C 180,E1 -22847.622,E2 -22847.622} C_VEL
LIN {X 0,Y 205.923,Z 497.48,A -85,B 0,C 180,E1 -22851.165,E2 -22851.165} C_VEL
LIN {X 0,Y 204.106,Z 503.645,A -85,B 0,C 180,E1 -22853.574,E2 -22853.574} C_VEL
LIN {X 0,Y 197.679,Z 513.095,A -85,B 0,C 180,E1 -22856.394,E2 -22856.394} C_VEL
LIN {X 0,Y 191.595,Z 520.866,A -85,B 0,C 180,E1 -22859.474,E2 -22859.474} C_VEL
LIN {X 0,Y 187.043,Z 526.038,A -85,B 0,C 180,E1 -22862.153,E2 -22862.153} C_VEL
LIN {X 0,Y 182.246,Z 530.982,A -85,B 0,C 180,E1 -22865.58,E2 -22865.58} C_VEL
LIN {X 0,Y 178.056,Z 534.807,A -85,B 0,C 180,E1 -22869.309,E2 -22869.309} C_VEL
LIN {X 0,Y 176,Z 536.412,A -85,B 0,C 180,E1 -22871.516,E2 -22871.516} C_VEL
LIN {X 0,Y 173.917,Z 537.761,A -85,B 0,C 180,E1 -22874.091,E2 -22874.091} C_VEL
LIN {X 0,Y 172.303,Z 538.608,A -85,B 0,C 180,E1 -22876.589,E2 -22876.589} C_VEL
LIN {X 0,Y 170.978,Z 538.986,A -85,B 0,C 180,E1 -22879.197,E2 -22879.197} C_VEL
LIN {X 0,Y 169.305,Z 538.479,A -85,B 0,C 180,E1 -22884.033,E2 -22884.033} C_VEL
LIN {X 0,Y 168.524,Z 536.397,A -85,B 0,C 180,E1 -22888.856,E2 -22888.856} C_VEL
LIN {X 0,Y 168.555,Z 532.865,A -85,B 0,C 180,E1 -22893.49,E2 -22893.49} C_VEL
LIN {X 0,Y 168.966,Z 529.345,A -85,B 0,C 180,E1 -22896.754,E2 -22896.754} C_VEL
LIN {X 0,Y 169.765,Z 523.854,A -85,B 0,C 180,E1 -22900.693,E2 -22900.693} C_VEL
LIN {X 0,Y 170.808,Z 517.215,A -85,B 0,C 180,E1 -22904.384,E2 -22904.384} C_VEL
LIN {X 0,Y 172.327,Z 509.329,A -85,B 0,C 180,E1 -22907.866,E2 -22907.866} C_VEL
LIN {X 0,Y 174.105,Z 500.556,A -85,B 0,C 180,E1 -22910.99,E2 -22910.99} C_VEL
LIN {X 0,Y 176.196,Z 490.436,A -85,B 0,C 180,E1 -22913.872,E2 -22913.872} C_VEL
LIN {X 0,Y 178.509,Z 478.604,A -85,B 0,C 180,E1 -22916.546,E2 -22916.546} C_VEL
LIN {X 0,Y 178.665,Z 475.072,A -85,B 0,C 180,E1 -22917.252,E2 -22917.252} C_VEL
LIN {X 0,Y 177.459,Z 464.029,A -85,B 0,C 180,E1 -22919.338,E2 -22919.338} C_VEL
LIN {X 0,Y 175.728,Z 451.242,A -85,B 0,C 180,E1 -22921.315,E2 -22921.315} C_VEL
LIN {X 0,Y 173.494,Z 438.007,A -85,B 0,C 180,E1 -22922.965,E2 -22922.965} C_VEL
LIN {X 0,Y 172.168,Z 430.803,A -85,B 0,C 180,E1 -22923.752,E2 -22923.752} C_VEL
LIN {X 0,Y 172.694,Z 426.673,A -85,B 0,C 180,E1 -22927.251,E2 -22927.251} C_VEL
LIN {X 0,Y 172.548,Z 424.115,A -85,B 0,C 180,E1 -22929.519,E2 -22929.519} C_VEL
LIN {X 0,Y 171.673,Z 419.101,A -85,B 0,C 180,E1 -22934.258,E2 -22934.258} C_VEL
LIN {X 0,Y 171.668,Z 419.286,A -85,B 0,C 180,E1 -22936.38,E2 -22936.38} C_VEL
LIN {X 0,Y 172.285,Z 422.112,A -85,B 0,C 180,E1 -22940.604,E2 -22940.604} C_VEL
LIN {X 0,Y 172.889,Z 425.472,A -85,B 0,C 180,E1 -22945.332,E2 -22945.332} C_VEL
LIN {X 0,Y 173.262,Z 427.213,A -85,B 0,C 180,E1 -22947.67,E2 -22947.67} C_VEL
LIN {X 0,Y 172.438,Z 430.253,A -85,B 0,C 180,E1 -22951.381,E2 -22951.381} C_VEL
LIN {X 0,Y 175.337,Z 442.095,A -85,B 0,C 180,E1 -22952.987,E2 -22952.987} C_VEL
LIN {X 0,Y 177.433,Z 453.506,A -85,B 0,C 180,E1 -22954.828,E2 -22954.828} C_VEL
LIN {X 0,Y 178.78,Z 464.58,A -85,B 0,C 180,E1 -22956.977,E2 -22956.977} C_VEL
LIN {X 0,Y 179.337,Z 471.965,A -85,B 0,C 180,E1 -22958.655,E2 -22958.655} C_VEL
LIN {X 0,Y 178.407,Z 477.76,A -85,B 0,C 180,E1 -22959.999,E2 -22959.999} C_VEL
LIN {X 0,Y 176.199,Z 487.347,A -85,B 0,C 180,E1 -22962.667,E2 -22962.667} C_VEL
LIN {X 0,Y 174.137,Z 495.608,A -85,B 0,C 180,E1 -22965.593,E2 -22965.593} C_VEL
LIN {X 0,Y 172.258,Z 503.153,A -85,B 0,C 180,E1 -22969.044,E2 -22969.044} C_VEL
LIN {X 0,Y 171.114,Z 507.708,A -85,B 0,C 180,E1 -22971.688,E2 -22971.688} C_VEL
LIN {X 0,Y 169.924,Z 513.118,A -85,B 0,C 180,E1 -22975.795,E2 -22975.795} C_VEL
LIN {X 0,Y 169.202,Z 516.842,A -85,B 0,C 180,E1 -22979.89,E2 -22979.89} C_VEL
LIN {X 0,Y 169.128,Z 518.97,A -85,B 0,C 180,E1 -22983.791,E2 -22983.791} C_VEL
LIN {X 0,Y 169.777,Z 519.905,A -85,B 0,C 180,E1 -22988.376,E2 -22988.376} C_VEL
LIN {X 0,Y 170.949,Z 519.338,A -85,B 0,C 180,E1 -22992.269,E2 -22992.269} C_VEL
LIN {X 0,Y 172.888,Z 517.43,A -85,B 0,C 180,E1 -22996.287,E2 -22996.287} C_VEL
LIN {X 0,Y 175.339,Z 514.161,A -85,B 0,C 180,E1 -23000.111,E2 -23000.111} C_VEL
LIN {X 0,Y 178.436,Z 509.502,A -85,B 0,C 180,E1 -23003.787,E2 -23003.787} C_VEL
LIN {X 0,Y 182.291,Z 503.091,A -85,B 0,C 180,E1 -23007.334,E2 -23007.334} C_VEL
LIN {X 0,Y 186.148,Z 495.952,A -85,B 0,C 180,E1 -23010.257,E2 -23010.257} C_VEL
LIN {X 0,Y 189.808,Z 488.273,A -85,B 0,C 180,E1 -23012.691,E2 -23012.691} C_VEL
LIN {X 0,Y 190.709,Z 483.336,A -85,B 0,C 180,E1 -23014.342,E2 -23014.342} C_VEL
LIN {X 0,Y 190.824,Z 475.267,A -85,B 0,C 180,E1 -23017.02,E2 -23017.02} C_VEL
LIN {X 0,Y 190.066,Z 466.93,A -85,B 0,C 180,E1 -23019.686,E2 -23019.686} C_VEL
LIN {X 0,Y 188.563,Z 459.715,A -85,B 0,C 180,E1 -23022.093,E2 -23022.093} C_VEL
LIN {X 0,Y 186.855,Z 454.788,A -85,B 0,C 180,E1 -23023.896,E2 -23023.896} C_VEL
LIN {X 0,Y 183.696,Z 448.051,A -85,B 0,C 180,E1 -23026.73,E2 -23026.73} C_VEL
LIN {X 0,Y 181.244,Z 443.532,A -85,B 0,C 180,E1 -23028.821,E2 -23028.821} C_VEL
LIN {X 0,Y 179.072,Z 439.976,A -85,B 0,C 180,E1 -23030.684,E2 -23030.684} C_VEL
LIN {X 0,Y 178.524,Z 438.789,A -85,B 0,C 180,E1 -23031.226,E2 -23031.226} C_VEL
LIN {X 0,Y 176.036,Z 435.998,A -85,B 0,C 180,E1 -23033.266,E2 -23033.266} C_VEL
LIN {X 0,Y 174.823,Z 433.249,A -85,B 0,C 180,E1 -23034.667,E2 -23034.667} C_VEL
LIN {X 0,Y 174.998,Z 431.715,A -85,B 0,C 180,E1 -23040.001,E2 -23040.001} C_VEL
LIN {X 0,Y 174.559,Z 431.044,A -85,B 0,C 180,E1 -23044.619,E2 -23044.619} C_VEL
LIN {X 0,Y 174.429,Z 430.687,A -85,B 0,C 180,E1 -23049.275,E2 -23049.275} C_VEL
LIN {X 0,Y 174.275,Z 430.852,A -85,B 0,C 180,E1 -23054.594,E2 -23054.594} C_VEL
LIN {X 0,Y 174.343,Z 431.35,A -85,B 0,C 180,E1 -23058.815,E2 -23058.815} C_VEL
LIN {X 0,Y 174.444,Z 432.013,A -85,B 0,C 180,E1 -23062.102,E2 -23062.102} C_VEL
LIN {X 0,Y 174.678,Z 433.684,A -85,B 0,C 180,E1 -23067.744,E2 -23067.744} C_VEL
LIN {X 0,Y 175.022,Z 435.571,A -85,B 0,C 180,E1 -23072.526,E2 -23072.526} C_VEL
LIN {X 0,Y 175.429,Z 437.495,A -85,B 0,C 180,E1 -23076.044,E2 -23076.044} C_VEL
LIN {X 0,Y 176.897,Z 440.671,A -85,B 0,C 180,E1 -23077.464,E2 -23077.464} C_VEL
LIN {X 0,Y 179.593,Z 444.107,A -85,B 0,C 180,E1 -23079.572,E2 -23079.572} C_VEL
LIN {X 0,Y 181.693,Z 448.117,A -85,B 0,C 180,E1 -23081.3,E2 -23081.3} C_VEL
LIN {X 0,Y 183.106,Z 449.991,A -85,B 0,C 180,E1 -23082.291,E2 -23082.291} C_VEL
LIN {X 0,Y 187.808,Z 459.741,A -85,B 0,C 180,E1 -23086.017,E2 -23086.017} C_VEL
LIN {X 0,Y 191.063,Z 468.483,A -85,B 0,C 180,E1 -23088.943,E2 -23088.943} C_VEL
LIN {X 0,Y 191.82,Z 471.78,A -85,B 0,C 180,E1 -23089.893,E2 -23089.893} C_VEL
LIN {X 0,Y 191.631,Z 482.577,A -85,B 0,C 180,E1 -23092.44,E2 -23092.44} C_VEL
LIN {X 0,Y 190.465,Z 491.857,A -85,B 0,C 180,E1 -23094.778,E2 -23094.778} C_VEL
LIN {X 0,Y 188.408,Z 500.848,A -85,B 0,C 180,E1 -23097.263,E2 -23097.263} C_VEL
LIN {X 0,Y 185.48,Z 507.591,A -85,B 0,C 180,E1 -23099.241,E2 -23099.241} C_VEL
LIN {X 0,Y 181.83,Z 514.722,A -85,B 0,C 180,E1 -23101.746,E2 -23101.746} C_VEL
LIN {X 0,Y 178.728,Z 520.61,A -85,B 0,C 180,E1 -23104.377,E2 -23104.377} C_VEL
LIN {X 0,Y 175.712,Z 526.357,A -85,B 0,C 180,E1 -23107.674,E2 -23107.674} C_VEL
LIN {X 0,Y 173.158,Z 530.858,A -85,B 0,C 180,E1 -23111.059,E2 -23111.059} C_VEL
LIN {X 0,Y 171.706,Z 533.243,A -85,B 0,C 180,E1 -23113.357,E2 -23113.357} C_VEL
LIN {X 0,Y 170.6,Z 535.198,A -85,B 0,C 180,E1 -23115.695,E2 -23115.695} C_VEL
LIN {X 0,Y 169.886,Z 536.681,A -85,B 0,C 180,E1 -23118.068,E2 -23118.068} C_VEL
LIN {X 0,Y 169.143,Z 538.428,A -85,B 0,C 180,E1 -23122.845,E2 -23122.845} C_VEL
LIN {X 0,Y 169.15,Z 538.735,A -85,B 0,C 180,E1 -23124.641,E2 -23124.641} C_VEL
LIN {X 0,Y 169.125,Z 541.796,A -85,B 0,C 180,E1 -23127.64,E2 -23127.64} C_VEL
LIN {X 0,Y 169.29,Z 543.683,A -85,B 0,C 180,E1 -23130.005,E2 -23130.005} C_VEL
LIN {X 0,Y 168.983,Z 545.622,A -85,B 0,C 180,E1 -23133.466,E2 -23133.466} C_VEL
LIN {X 0,Y 169.161,Z 546.837,A -85,B 0,C 180,E1 -23137.728,E2 -23137.728} C_VEL
LIN {X 0,Y 168.828,Z 547.02,A -85,B 0,C 180,E1 -23139.73,E2 -23139.73} C_VEL
LIN {X 0,Y 166.892,Z 546.746,A -85,B 0,C 180,E1 -23143.056,E2 -23143.056} C_VEL
LIN {X 0,Y 165.547,Z 545.94,A -85,B 0,C 180,E1 -23146.435,E2 -23146.435} C_VEL
LIN {X 0,Y 166.134,Z 545.123,A -85,B 0,C 180,E1 -23148.448,E2 -23148.448} C_VEL
LIN {X 0,Y 169.011,Z 543.073,A -85,B 0,C 180,E1 -23151.983,E2 -23151.983} C_VEL
LIN {X 0,Y 173.766,Z 538.93,A -85,B 0,C 180,E1 -23156.422,E2 -23156.422} C_VEL
LIN {X 0,Y 178.161,Z 534.505,A -85,B 0,C 180,E1 -23159.789,E2 -23159.789} C_VEL
LIN {X 0,Y 182.69,Z 529.618,A -85,B 0,C 180,E1 -23162.592,E2 -23162.592} C_VEL
LIN {X 0,Y 189.135,Z 522.089,A -85,B 0,C 180,E1 -23165.825,E2 -23165.825} C_VEL
LIN {X 0,Y 196.239,Z 512.674,A -85,B 0,C 180,E1 -23168.814,E2 -23168.814} C_VEL
LIN {X 0,Y 201.016,Z 503.548,A -85,B 0,C 180,E1 -23171.632,E2 -23171.632} C_VEL
LIN {X 0,Y 203.851,Z 496.777,A -85,B 0,C 180,E1 -23173.613,E2 -23173.613} C_VEL
LIN {X 0,Y 204.398,Z 495.109,A -85,B 0,C 180,E1 -23174.159,E2 -23174.159} C_VEL
LIN {X 0,Y 204.331,Z 490.548,A -85,B 0,C 180,E1 -23176.535,E2 -23176.535} C_VEL
LIN {X 0,Y 203.955,Z 486.215,A -85,B 0,C 180,E1 -23179.301,E2 -23179.301} C_VEL
LIN {X 0,Y 203.379,Z 483.661,A -85,B 0,C 180,E1 -23181.536,E2 -23181.536} C_VEL
LIN {X 0,Y 202.121,Z 480.265,A -85,B 0,C 180,E1 -23186.571,E2 -23186.571} C_VEL
LIN {X 0,Y 201.844,Z 479.603,A -85,B 0,C 180,E1 -23188.514,E2 -23188.514} C_VEL
LIN {X 0,Y 201.679,Z 479.31,A -85,B 0,C 180,E1 -23190.799,E2 -23190.799} C_VEL
LIN {X 0,Y 201.593,Z 479.677,A -85,B 0,C 180,E1 -23193.049,E2 -23193.049} C_VEL
LIN {X 0,Y 201.823,Z 481.861,A -85,B 0,C 180,E1 -23197.477,E2 -23197.477} C_VEL
LIN {X 0,Y 202.211,Z 483.581,A -85,B 0,C 180,E1 -23199.794,E2 -23199.794} C_VEL
LIN {X 0,Y 202.621,Z 486.803,A -85,B 0,C 180,E1 -23202.754,E2 -23202.754} C_VEL
LIN {X 0,Y 202.952,Z 491.348,A -85,B 0,C 180,E1 -23205.971,E2 -23205.971} C_VEL
LIN {X 0,Y 202.44,Z 494.438,A -85,B 0,C 180,E1 -23207.468,E2 -23207.468} C_VEL
LIN {X 0,Y 200.132,Z 502.429,A -85,B 0,C 180,E1 -23210.907,E2 -23210.907} C_VEL
LIN {X 0,Y 199.292,Z 504.748,A -85,B 0,C 180,E1 -23211.89,E2 -23211.89} C_VEL
LIN {X 0,Y 198.482,Z 506.469,A -85,B 0,C 180,E1 -23212.523,E2 -23212.523} C_VEL
LIN {X 0,Y 191.936,Z 515.136,A -85,B 0,C 180,E1 -23215.274,E2 -23215.274} C_VEL
LIN {X 0,Y 185.669,Z 522.446,A -85,B 0,C 180,E1 -23218.372,E2 -23218.372} C_VEL
LIN {X 0,Y 180.939,Z 527.368,A -85,B 0,C 180,E1 -23221.112,E2 -23221.112} C_VEL
LIN {X 0,Y 175.973,Z 532.004,A -85,B 0,C 180,E1 -23224.581,E2 -23224.581} C_VEL
LIN {X 0,Y 170.845,Z 536.033,A -85,B 0,C 180,E1 -23229.125,E2 -23229.125} C_VEL
LIN {X 0,Y 168.19,Z 537.725,A -85,B 0,C 180,E1 -23232.059,E2 -23232.059} C_VEL
LIN {X 0,Y 166.243,Z 538.676,A -85,B 0,C 180,E1 -23234.693,E2 -23234.693} C_VEL
LIN {X 0,Y 163.79,Z 539.246,A -85,B 0,C 180,E1 -23239.255,E2 -23239.255} C_VEL
LIN {X 0,Y 162.087,Z 538.281,A -85,B 0,C 180,E1 -23244.409,E2 -23244.409} C_VEL
LIN {X 0,Y 161.385,Z 535.809,A -85,B 0,C 180,E1 -23249.421,E2 -23249.421} C_VEL
LIN {X 0,Y 161.405,Z 533.124,A -85,B 0,C 180,E1 -23252.875,E2 -23252.875} C_VEL
LIN {X 0,Y 161.972,Z 528.324,A -85,B 0,C 180,E1 -23257.405,E2 -23257.405} C_VEL
LIN {X 0,Y 162.904,Z 522.181,A -85,B 0,C 180,E1 -23261.683,E2 -23261.683} C_VEL
LIN {X 0,Y 164.247,Z 514.554,A -85,B 0,C 180,E1 -23265.783,E2 -23265.783} C_VEL
LIN {X 0,Y 166.025,Z 505.337,A -85,B 0,C 180,E1 -23269.636,E2 -23269.636} C_VEL
LIN {X 0,Y 167.98,Z 496.329,A -85,B 0,C 180,E1 -23272.647,E2 -23272.647} C_VEL
LIN {X 0,Y 170.307,Z 485.128,A -85,B 0,C 180,E1 -23275.621,E2 -23275.621} C_VEL
LIN {X 0,Y 171.693,Z 478.178,A -85,B 0,C 180,E1 -23277.15,E2 -23277.15} C_VEL
LIN {X 0,Y 170.989,Z 468.856,A -85,B 0,C 180,E1 -23279.08,E2 -23279.08} C_VEL
LIN {X 0,Y 169.548,Z 456.843,A -85,B 0,C 180,E1 -23281.187,E2 -23281.187} C_VEL
LIN {X 0,Y 167.497,Z 443.541,A -85,B 0,C 180,E1 -23283.105,E2 -23283.105} C_VEL
LIN {X 0,Y 165.213,Z 431.025,A -85,B 0,C 180,E1 -23284.514,E2 -23284.514} C_VEL
LIN {X 0,Y 165.68,Z 427.542,A -85,B 0,C 180,E1 -23287.551,E2 -23287.551} C_VEL
LIN {X 0,Y 165.432,Z 424.723,A -85,B 0,C 180,E1 -23290.126,E2 -23290.126} C_VEL
LIN {X 0,Y 164.608,Z 419.981,A -85,B 0,C 180,E1 -23294.677,E2 -23294.677} C_VEL
LIN {X 0,Y 164.608,Z 419.993,A -85,B 0,C 180,E1 -23295.152,E2 -23295.152} C_VEL
LIN {X 0,Y 165.257,Z 423.229,A -85,B 0,C 180,E1 -23300.201,E2 -23300.201} C_VEL
LIN {X 0,Y 165.877,Z 426.603,A -85,B 0,C 180,E1 -23305.134,E2 -23305.134} C_VEL
LIN {X 0,Y 166.26,Z 428.349,A -85,B 0,C 180,E1 -23307.572,E2 -23307.572} C_VEL
LIN {X 0,Y 165.633,Z 430.522,A -85,B 0,C 180,E1 -23310.299,E2 -23310.299} C_VEL
LIN {X 0,Y 168.665,Z 443.113,A -85,B 0,C 180,E1 -23312.067,E2 -23312.067} C_VEL
LIN {X 0,Y 170.56,Z 453.325,A -85,B 0,C 180,E1 -23313.799,E2 -23313.799} C_VEL
LIN {X 0,Y 171.984,Z 464.986,A -85,B 0,C 180,E1 -23316.168,E2 -23316.168} C_VEL
LIN {X 0,Y 172.526,Z 473.462,A -85,B 0,C 180,E1 -23318.191,E2 -23318.191} C_VEL
LIN {X 0,Y 170.639,Z 482.375,A -85,B 0,C 180,E1 -23320.462,E2 -23320.462} C_VEL
LIN {X 0,Y 168.442,Z 491.144,A -85,B 0,C 180,E1 -23323.261,E2 -23323.261} C_VEL
LIN {X 0,Y 166.682,Z 497.967,A -85,B 0,C 180,E1 -23325.984,E2 -23325.984} C_VEL
LIN {X 0,Y 164.999,Z 504.503,A -85,B 0,C 180,E1 -23329.269,E2 -23329.269} C_VEL
LIN {X 0,Y 163.622,Z 509.872,A -85,B 0,C 180,E1 -23332.735,E2 -23332.735} C_VEL
LIN {X 0,Y 162.877,Z 513.29,A -85,B 0,C 180,E1 -23335.556,E2 -23335.556} C_VEL
LIN {X 0,Y 162.11,Z 517.13,A -85,B 0,C 180,E1 -23339.883,E2 -23339.883} C_VEL
LIN {X 0,Y 162.075,Z 519.524,A -85,B 0,C 180,E1 -23344.525,E2 -23344.525} C_VEL
LIN {X 0,Y 162.811,Z 520.327,A -85,B 0,C 180,E1 -23349.015,E2 -23349.015} C_VEL
LIN {X 0,Y 164.265,Z 519.669,A -85,B 0,C 180,E1 -23353.338,E2 -23353.338} C_VEL
LIN {X 0,Y 166.411,Z 517.648,A -85,B 0,C 180,E1 -23357.491,E2 -23357.491} C_VEL
LIN {X 0,Y 169.092,Z 514.307,A -85,B 0,C 180,E1 -23361.433,E2 -23361.433} C_VEL
LIN {X 0,Y 172.521,Z 509.494,A -85,B 0,C 180,E1 -23365.229,E2 -23365.229} C_VEL
LIN {X 0,Y 175.821,Z 504.346,A -85,B 0,C 180,E1 -23368.198,E2 -23368.198} C_VEL
LIN {X 0,Y 180.118,Z 497.017,A -85,B 0,C 180,E1 -23371.38,E2 -23371.38} C_VEL
LIN {X 0,Y 184.089,Z 488.925,A -85,B 0,C 180,E1 -23374.066,E2 -23374.066} C_VEL
LIN {X 0,Y 184.954,Z 482.875,A -85,B 0,C 180,E1 -23376.247,E2 -23376.247} C_VEL
LIN {X 0,Y 184.95,Z 473.88,A -85,B 0,C 180,E1 -23379.422,E2 -23379.422} C_VEL
LIN {X 0,Y 184.295,Z 467.459,A -85,B 0,C 180,E1 -23381.664,E2 -23381.664} C_VEL
LIN {X 0,Y 183.166,Z 462.321,A -85,B 0,C 180,E1 -23383.563,E2 -23383.563} C_VEL
LIN {X 0,Y 180.65,Z 455.541,A -85,B 0,C 180,E1 -23386.502,E2 -23386.502} C_VEL
LIN {X 0,Y 177.929,Z 449.613,A -85,B 0,C 180,E1 -23389.331,E2 -23389.331} C_VEL
LIN {X 0,Y 175.269,Z 444.759,A -85,B 0,C 180,E1 -23392.047,E2 -23392.047} C_VEL
LIN {X 0,Y 173.047,Z 441.692,A -85,B 0,C 180,E1 -23394.246,E2 -23394.246} C_VEL
LIN {X 0,Y 172.085,Z 439.565,A -85,B 0,C 180,E1 -23395.462,E2 -23395.462} C_VEL
LIN {X 0,Y 169.62,Z 436.992,A -85,B 0,C 180,E1 -23398.116,E2 -23398.116} C_VEL
LIN {X 0,Y 168.199,Z 433.808,A -85,B 0,C 180,E1 -23400.45,E2 -23400.45} C_VEL
LIN {X 0,Y 167.806,Z 433.268,A -85,B 0,C 180,E1 -23404.806,E2 -23404.806} C_VEL
LIN {X 0,Y 167.686,Z 432.972,A -85,B 0,C 180,E1 -23409.652,E2 -23409.652} C_VEL
LIN {X 0,Y 167.556,Z 433.205,A -85,B 0,C 180,E1 -23415.291,E2 -23415.291} C_VEL
LIN {X 0,Y 167.642,Z 433.785,A -85,B 0,C 180,E1 -23419.597,E2 -23419.597} C_VEL
LIN {X 0,Y 167.714,Z 434.461,A -85,B 0,C 180,E1 -23422.811,E2 -23422.811} C_VEL
LIN {X 0,Y 168.005,Z 436.199,A -85,B 0,C 180,E1 -23428.555,E2 -23428.555} C_VEL
LIN {X 0,Y 168.099,Z 436.867,A -85,B 0,C 180,E1 -23429.849,E2 -23429.849} C_VEL
LIN {X 0,Y 170.081,Z 440.704,A -85,B 0,C 180,E1 -23432.493,E2 -23432.493} C_VEL
LIN {X 0,Y 172.758,Z 443.783,A -85,B 0,C 180,E1 -23435.216,E2 -23435.216} C_VEL
LIN {X 0,Y 174.43,Z 447.343,A -85,B 0,C 180,E1 -23437.044,E2 -23437.044} C_VEL
LIN {X 0,Y 176.369,Z 450.079,A -85,B 0,C 180,E1 -23438.784,E2 -23438.784} C_VEL
LIN {X 0,Y 178.25,Z 453.905,A -85,B 0,C 180,E1 -23440.585,E2 -23440.585} C_VEL
LIN {X 0,Y 179.932,Z 457.085,A -85,B 0,C 180,E1 -23442.096,E2 -23442.096} C_VEL
LIN {X 0,Y 181.996,Z 461.664,A -85,B 0,C 180,E1 -23444.036,E2 -23444.036} C_VEL
LIN {X 0,Y 184.422,Z 467.776,A -85,B 0,C 180,E1 -23446.391,E2 -23446.391} C_VEL
LIN {X 0,Y 186.377,Z 474.163,A -85,B 0,C 180,E1 -23448.636,E2 -23448.636} C_VEL
LIN {X 0,Y 186.017,Z 483.833,A -85,B 0,C 180,E1 -23451.112,E2 -23451.112} C_VEL
LIN {X 0,Y 184.609,Z 493.046,A -85,B 0,C 180,E1 -23453.576,E2 -23453.576} C_VEL
LIN {X 0,Y 182.441,Z 501.434,A -85,B 0,C 180,E1 -23456.05,E2 -23456.05} C_VEL
LIN {X 0,Y 179.449,Z 508.033,A -85,B 0,C 180,E1 -23458.088,E2 -23458.088} C_VEL
LIN {X 0,Y 174.927,Z 516.223,A -85,B 0,C 180,E1 -23461.183,E2 -23461.183} C_VEL
LIN {X 0,Y 171.253,Z 522.644,A -85,B 0,C 180,E1 -23464.385,E2 -23464.385} C_VEL
LIN {X 0,Y 168.135,Z 528.002,A -85,B 0,C 180,E1 -23467.908,E2 -23467.908} C_VEL
LIN {X 0,Y 165.619,Z 532.026,A -85,B 0,C 180,E1 -23471.448,E2 -23471.448} C_VEL
LIN {X 0,Y 163.686,Z 534.992,A -85,B 0,C 180,E1 -23475.077,E2 -23475.077} C_VEL
LIN {X 0,Y 162.358,Z 537.438,A -85,B 0,C 180,E1 -23480.035,E2 -23480.035} C_VEL
LIN {X 0,Y 162.085,Z 538.349,A -85,B 0,C 180,E1 -23484.875,E2 -23484.875} C_VEL
LIN {X 0,Y 162.097,Z 542.077,A -85,B 0,C 180,E1 -23488.763,E2 -23488.763} C_VEL
LIN {X 0,Y 162.228,Z 543.041,A -85,B 0,C 180,E1 -23490.006,E2 -23490.006} C_VEL
LIN {X 0,Y 161.917,Z 544.986,A -85,B 0,C 180,E1 -23493.311,E2 -23493.311} C_VEL
LIN {X 0,Y 162.079,Z 546.477,A -85,B 0,C 180,E1 -23497.839,E2 -23497.839} C_VEL
LIN {X 0,Y 163.166,Z 546.761,A -85,B 0,C 180,E1 -23502.442,E2 -23502.442} C_VEL
LIN {X 0,Y 165.375,Z 545.643,A -85,B 0,C 180,E1 -23507.312,E2 -23507.312} C_VEL
LIN {X 0,Y 166.134,Z 545.123,A -85,B 0,C 180,E1 -23508.448,E2 -23508.448} C_VEL
LIN {X 0,Y 166.985,Z 544.189,A -85,B 0,C 180,E1 -23510.433,E2 -23510.433} C_VEL
LIN {X 0,Y 167.13,Z 542.313,A -85,B 0,C 180,E1 -23513.773,E2 -23513.773} C_VEL
LIN {X 0,Y 167.461,Z 540.407,A -85,B 0,C 180,E1 -23516.413,E2 -23516.413} C_VEL
LIN {X 0,Y 168.596,Z 538.633,A -85,B 0,C 180,E1 -23518.299,E2 -23518.299} C_VEL
LIN {X 0,Y 169.237,Z 537.966,A -85,B 0,C 180,E1 -23518.89,E2 -23518.89} C_VEL
LIN {X 0,Y 175.061,Z 532.422,A -85,B 0,C 180,E1 -23522.823,E2 -23522.823} C_VEL
LIN {X 0,Y 181.582,Z 525.731,A -85,B 0,C 180,E1 -23526.179,E2 -23526.179} C_VEL
LIN {X 0,Y 187.712,Z 518.665,A -85,B 0,C 180,E1 -23528.843,E2 -23528.843} C_VEL
LIN {X 0,Y 191.847,Z 513.167,A -85,B 0,C 180,E1 -23530.565,E2 -23530.565} C_VEL
LIN {X 0,Y 196.923,Z 504.257,A -85,B 0,C 180,E1 -23533.441,E2 -23533.441} C_VEL
LIN {X 0,Y 199.425,Z 498.803,A -85,B 0,C 180,E1 -23535.184,E2 -23535.184} C_VEL
LIN {X 0,Y 199.629,Z 493.985,A -85,B 0,C 180,E1 -23538.017,E2 -23538.017} C_VEL
LIN {X 0,Y 199.377,Z 490.202,A -85,B 0,C 180,E1 -23540.855,E2 -23540.855} C_VEL
LIN {X 0,Y 198.462,Z 487.404,A -85,B 0,C 180,E1 -23544.542,E2 -23544.542} C_VEL
LIN {X 0,Y 197.991,Z 485.59,A -85,B 0,C 180,E1 -23548.427,E2 -23548.427} C_VEL
LIN {X 0,Y 197.854,Z 485.335,A -85,B 0,C 180,E1 -23550.178,E2 -23550.178} C_VEL
LIN {X 0,Y 197.711,Z 485.552,A -85,B 0,C 180,E1 -23552.714,E2 -23552.714} C_VEL
LIN {X 0,Y 197.735,Z 487.805,A -85,B 0,C 180,E1 -23557.542,E2 -23557.542} C_VEL
LIN {X 0,Y 197.929,Z 489.685,A -85,B 0,C 180,E1 -23560.022,E2 -23560.022} C_VEL
LIN {X 0,Y 198.09,Z 493.465,A -85,B 0,C 180,E1 -23563.51,E2 -23563.51} C_VEL
LIN {X 0,Y 197.918,Z 496.493,A -85,B 0,C 180,E1 -23565.607,E2 -23565.607} C_VEL
LIN {X 0,Y 196.605,Z 500.628,A -85,B 0,C 180,E1 -23567.614,E2 -23567.614} C_VEL
LIN {X 0,Y 194.13,Z 507.141,A -85,B 0,C 180,E1 -23570.623,E2 -23570.623} C_VEL
LIN {X 0,Y 193.476,Z 508.33,A -85,B 0,C 180,E1 -23571.118,E2 -23571.118} C_VEL
LIN {X 0,Y 186.466,Z 516.967,A -85,B 0,C 180,E1 -23574.018,E2 -23574.018} C_VEL
LIN {X 0,Y 179.827,Z 524.007,A -85,B 0,C 180,E1 -23577.199,E2 -23577.199} C_VEL
LIN {X 0,Y 174.868,Z 528.659,A -85,B 0,C 180,E1 -23579.999,E2 -23579.999} C_VEL
LIN {X 0,Y 169.093,Z 533.448,A -85,B 0,C 180,E1 -23583.989,E2 -23583.989} C_VEL
LIN {X 0,Y 163.626,Z 537.156,A -85,B 0,C 180,E1 -23588.901,E2 -23588.901} C_VEL
LIN {X 0,Y 159.395,Z 539.12,A -85,B 0,C 180,E1 -23594.049,E2 -23594.049} C_VEL
LIN {X 0,Y 156.534,Z 539.353,A -85,B 0,C 180,E1 -23599.451,E2 -23599.451} C_VEL
LIN {X 0,Y 154.875,Z 537.978,A -85,B 0,C 180,E1 -23604.817,E2 -23604.817} C_VEL
LIN {X 0,Y 154.267,Z 535.035,A -85,B 0,C 180,E1 -23610.074,E2 -23610.074} C_VEL
LIN {X 0,Y 154.548,Z 530.693,A -85,B 0,C 180,E1 -23615.053,E2 -23615.053} C_VEL
LIN {X 0,Y 155.314,Z 525.012,A -85,B 0,C 180,E1 -23619.706,E2 -23619.706} C_VEL
LIN {X 0,Y 156.474,Z 518.08,A -85,B 0,C 180,E1 -23624.051,E2 -23624.051} C_VEL
LIN {X 0,Y 158.116,Z 509.575,A -85,B 0,C 180,E1 -23628.179,E2 -23628.179} C_VEL
LIN {X 0,Y 160.062,Z 500.443,A -85,B 0,C 180,E1 -23631.706,E2 -23631.706} C_VEL
LIN {X 0,Y 162.289,Z 490.205,A -85,B 0,C 180,E1 -23634.822,E2 -23634.822} C_VEL
LIN {X 0,Y 164.579,Z 479.142,A -85,B 0,C 180,E1 -23637.511,E2 -23637.511} C_VEL
LIN {X 0,Y 164.707,Z 476.34,A -85,B 0,C 180,E1 -23638.123,E2 -23638.123} C_VEL
LIN {X 0,Y 163.448,Z 463.819,A -85,B 0,C 180,E1 -23640.713,E2 -23640.713} C_VEL
LIN {X 0,Y 161.944,Z 452.14,A -85,B 0,C 180,E1 -23642.685,E2 -23642.685} C_VEL
LIN {X 0,Y 159.663,Z 438.241,A -85,B 0,C 180,E1 -23644.579,E2 -23644.579} C_VEL
LIN {X 0,Y 158.312,Z 431.118,A -85,B 0,C 180,E1 -23645.4,E2 -23645.4} C_VEL
LIN {X 0,Y 158.631,Z 427.725,A -85,B 0,C 180,E1 -23648.492,E2 -23648.492} C_VEL
LIN {X 0,Y 157.943,Z 422.849,A -85,B 0,C 180,E1 -23653.183,E2 -23653.183} C_VEL
LIN {X 0,Y 157.637,Z 421.315,A -85,B 0,C 180,E1 -23654.81,E2 -23654.81} C_VEL
LIN {X 0,Y 158.229,Z 424.333,A -85,B 0,C 180,E1 -23659.761,E2 -23659.761} C_VEL
LIN {X 0,Y 158.586,Z 426.013,A -85,B 0,C 180,E1 -23662.354,E2 -23662.354} C_VEL
LIN {X 0,Y 159.252,Z 429.477,A -85,B 0,C 180,E1 -23667.465,E2 -23667.465} C_VEL
LIN {X 0,Y 158.855,Z 430.694,A -85,B 0,C 180,E1 -23669.044,E2 -23669.044} C_VEL
LIN {X 0,Y 162.066,Z 444.197,A -85,B 0,C 180,E1 -23671.113,E2 -23671.113} C_VEL
LIN {X 0,Y 163.702,Z 453.082,A -85,B 0,C 180,E1 -23672.706,E2 -23672.706} C_VEL
LIN {X 0,Y 165.025,Z 463.53,A -85,B 0,C 180,E1 -23674.881,E2 -23674.881} C_VEL
LIN {X 0,Y 165.725,Z 473.429,A -85,B 0,C 180,E1 -23677.304,E2 -23677.304} C_VEL
LIN {X 0,Y 164.915,Z 478.418,A -85,B 0,C 180,E1 -23678.572,E2 -23678.572} C_VEL
LIN {X 0,Y 162.668,Z 487.302,A -85,B 0,C 180,E1 -23681.205,E2 -23681.205} C_VEL
LIN {X 0,Y 160.368,Z 495.92,A -85,B 0,C 180,E1 -23684.446,E2 -23684.446} C_VEL
LIN {X 0,Y 158.351,Z 503.37,A -85,B 0,C 180,E1 -23688.094,E2 -23688.094} C_VEL
LIN {X 0,Y 156.826,Z 509.08,A -85,B 0,C 180,E1 -23691.691,E2 -23691.691} C_VEL
LIN {X 0,Y 155.758,Z 513.662,A -85,B 0,C 180,E1 -23695.523,E2 -23695.523} C_VEL
LIN {X 0,Y 155.004,Z 517.412,A -85,B 0,C 180,E1 -23699.91,E2 -23699.91} C_VEL
LIN {X 0,Y 154.895,Z 519.157,A -85,B 0,C 180,E1 -23702.981,E2 -23702.981} C_VEL
LIN {X 0,Y 155.151,Z 520.27,A -85,B 0,C 180,E1 -23706.069,E2 -23706.069} C_VEL
LIN {X 0,Y 155.968,Z 520.741,A -85,B 0,C 180,E1 -23710.003,E2 -23710.003} C_VEL
LIN {X 0,Y 157.623,Z 520.004,A -85,B 0,C 180,E1 -23714.489,E2 -23714.489} C_VEL
LIN {X 0,Y 159.972,Z 517.887,A -85,B 0,C 180,E1 -23718.778,E2 -23718.778} C_VEL
LIN {X 0,Y 162.934,Z 514.484,A -85,B 0,C 180,E1 -23722.853,E2 -23722.853} C_VEL
LIN {X 0,Y 166.707,Z 509.545,A -85,B 0,C 180,E1 -23726.767,E2 -23726.767} C_VEL
LIN {X 0,Y 170.498,Z 504.02,A -85,B 0,C 180,E1 -23729.942,E2 -23729.942} C_VEL
LIN {X 0,Y 174.171,Z 498.054,A -85,B 0,C 180,E1 -23732.575,E2 -23732.575} C_VEL
LIN {X 0,Y 178.103,Z 490.66,A -85,B 0,C 180,E1 -23735.159,E2 -23735.159} C_VEL
LIN {X 0,Y 179.152,Z 484.6,A -85,B 0,C 180,E1 -23737.513,E2 -23737.513} C_VEL
LIN {X 0,Y 179.408,Z 476.959,A -85,B 0,C 180,E1 -23740.432,E2 -23740.432} C_VEL
LIN {X 0,Y 178.851,Z 469.797,A -85,B 0,C 180,E1 -23743.155,E2 -23743.155} C_VEL
LIN {X 0,Y 177.506,Z 463.894,A -85,B 0,C 180,E1 -23745.674,E2 -23745.674} C_VEL
LIN {X 0,Y 175.357,Z 458.323,A -85,B 0,C 180,E1 -23748.441,E2 -23748.441} C_VEL
LIN {X 0,Y 173.583,Z 454.223,A -85,B 0,C 180,E1 -23750.681,E2 -23750.681} C_VEL
LIN {X 0,Y 171.719,Z 450.478,A -85,B 0,C 180,E1 -23752.948,E2 -23752.948} C_VEL
LIN {X 0,Y 168.974,Z 445.638,A -85,B 0,C 180,E1 -23756.466,E2 -23756.466} C_VEL
LIN {X 0,Y 166.546,Z 442.034,A -85,B 0,C 180,E1 -23759.871,E2 -23759.871} C_VEL
LIN {X 0,Y 166.059,Z 440.511,A -85,B 0,C 180,E1 -23760.91,E2 -23760.91} C_VEL
LIN {X 0,Y 161.809,Z 436.99,A -85,B 0,C 180,E1 -23770.006,E2 -23770.006} C_VEL
LIN {X 0,Y 161.398,Z 436.527,A -85,B 0,C 180,E1 -23772.576,E2 -23772.576} C_VEL
LIN {X 0,Y 161.326,Z 436.736,A -85,B 0,C 180,E1 -23776.607,E2 -23776.607} C_VEL
LIN {X 0,Y 162.005,Z 438.365,A -85,B 0,C 180,E1 -23780.972,E2 -23780.972} C_VEL
LIN {X 0,Y 165.95,Z 443.446,A -85,B 0,C 180,E1 -23789.141,E2 -23789.141} C_VEL
LIN {X 0,Y 168.212,Z 447.908,A -85,B 0,C 180,E1 -23792.544,E2 -23792.544} C_VEL
LIN {X 0,Y 169.852,Z 449.942,A -85,B 0,C 180,E1 -23794.434,E2 -23794.434} C_VEL
LIN {X 0,Y 171.894,Z 454.273,A -85,B 0,C 180,E1 -23796.943,E2 -23796.943} C_VEL
LIN {X 0,Y 173.107,Z 456.424,A -85,B 0,C 180,E1 -23798.254,E2 -23798.254} C_VEL
LIN {X 0,Y 175.85,Z 462.275,A -85,B 0,C 180,E1 -23801.256,E2 -23801.256} C_VEL
LIN {X 0,Y 178.581,Z 469.103,A -85,B 0,C 180,E1 -23804.312,E2 -23804.312} C_VEL
LIN {X 0,Y 180.97,Z 477.385,A -85,B 0,C 180,E1 -23807.551,E2 -23807.551} C_VEL
LIN {X 0,Y 180.751,Z 482.526,A -85,B 0,C 180,E1 -23808.992,E2 -23808.992} C_VEL
LIN {X 0,Y 179.353,Z 491.824,A -85,B 0,C 180,E1 -23811.602,E2 -23811.602} C_VEL
LIN {X 0,Y 177.158,Z 500.355,A -85,B 0,C 180,E1 -23814.194,E2 -23814.194} C_VEL
LIN {X 0,Y 175.172,Z 505.393,A -85,B 0,C 180,E1 -23815.835,E2 -23815.835} C_VEL
LIN {X 0,Y 170.256,Z 514.067,A -85,B 0,C 180,E1 -23818.943,E2 -23818.943} C_VEL
LIN {X 0,Y 166.011,Z 520.94,A -85,B 0,C 180,E1 -23822.253,E2 -23822.253} C_VEL
LIN {X 0,Y 162.642,Z 526.418,A -85,B 0,C 180,E1 -23825.77,E2 -23825.77} C_VEL
LIN {X 0,Y 159.717,Z 530.718,A -85,B 0,C 180,E1 -23829.395,E2 -23829.395} C_VEL
LIN {X 0,Y 158.101,Z 532.998,A -85,B 0,C 180,E1 -23831.877,E2 -23831.877} C_VEL
LIN {X 0,Y 156.796,Z 534.782,A -85,B 0,C 180,E1 -23834.405,E2 -23834.405} C_VEL
LIN {X 0,Y 155.322,Z 537.134,A -85,B 0,C 180,E1 -23839.579,E2 -23839.579} C_VEL
LIN {X 0,Y 155.005,Z 537.809,A -85,B 0,C 180,E1 -23844.803,E2 -23844.803} C_VEL
LIN {X 0,Y 155.167,Z 542.34,A -85,B 0,C 180,E1 -23850.006,E2 -23850.006} C_VEL
LIN {X 0,Y 154.859,Z 544.255,A -85,B 0,C 180,E1 -23853.192,E2 -23853.192} C_VEL
LIN {X 0,Y 154.985,Z 546.006,A -85,B 0,C 180,E1 -23857.824,E2 -23857.824} C_VEL
LIN {X 0,Y 156.234,Z 546.594,A -85,B 0,C 180,E1 -23863.004,E2 -23863.004} C_VEL
LIN {X 0,Y 158.59,Z 545.684,A -85,B 0,C 180,E1 -23868.077,E2 -23868.077} C_VEL
LIN {X 0,Y 162.464,Z 543.339,A -85,B 0,C 180,E1 -23872.918,E2 -23872.918} C_VEL
LIN {X 0,Y 167.453,Z 539.515,A -85,B 0,C 180,E1 -23877.5,E2 -23877.5} C_VEL
LIN {X 0,Y 169.237,Z 537.966,A -85,B 0,C 180,E1 -23878.89,E2 -23878.89} C_VEL
LIN {X 0,Y 170.915,Z 535.96,A -85,B 0,C 180,E1 -23880.675,E2 -23880.675} C_VEL
LIN {X 0,Y 172.603,Z 532.509,A -85,B 0,C 180,E1 -23883.729,E2 -23883.729} C_VEL
LIN {X 0,Y 174.82,Z 528.591,A -85,B 0,C 180,E1 -23886.615,E2 -23886.615} C_VEL
LIN {X 0,Y 177.232,Z 525.759,A -85,B 0,C 180,E1 -23888.092,E2 -23888.092} C_VEL
LIN {X 0,Y 184.622,Z 517.76,A -85,B 0,C 180,E1 -23891.051,E2 -23891.051} C_VEL
LIN {X 0,Y 188.558,Z 512.433,A -85,B 0,C 180,E1 -23892.866,E2 -23892.866} C_VEL
LIN {X 0,Y 193.438,Z 504.265,A -85,B 0,C 180,E1 -23895.588,E2 -23895.588} C_VEL
LIN {X 0,Y 194.417,Z 502.301,A -85,B 0,C 180,E1 -23896.306,E2 -23896.306} C_VEL
LIN {X 0,Y 194.82,Z 497.544,A -85,B 0,C 180,E1 -23899.507,E2 -23899.507} C_VEL
LIN {X 0,Y 194.825,Z 495.901,A -85,B 0,C 180,E1 -23900.872,E2 -23900.872} C_VEL
LIN {X 0,Y 194.207,Z 493.086,A -85,B 0,C 180,E1 -23904.618,E2 -23904.618} C_VEL
LIN {X 0,Y 193.905,Z 491.874,A -85,B 0,C 180,E1 -23907.066,E2 -23907.066} C_VEL
LIN {X 0,Y 193.661,Z 491.117,A -85,B 0,C 180,E1 -23910.578,E2 -23910.578} C_VEL
LIN {X 0,Y 193.556,Z 491.181,A -85,B 0,C 180,E1 -23911.833,E2 -23911.833} C_VEL
LIN {X 0,Y 193.327,Z 492.832,A -85,B 0,C 180,E1 -23916.428,E2 -23916.428} C_VEL
LIN {X 0,Y 193.384,Z 494.188,A -85,B 0,C 180,E1 -23918.689,E2 -23918.689} C_VEL
LIN {X 0,Y 193.278,Z 497.239,A -85,B 0,C 180,E1 -23921.996,E2 -23921.996} C_VEL
LIN {X 0,Y 193.06,Z 499.79,A -85,B 0,C 180,E1 -23924.155,E2 -23924.155} C_VEL
LIN {X 0,Y 192.644,Z 501.415,A -85,B 0,C 180,E1 -23925.204,E2 -23925.204} C_VEL
LIN {X 0,Y 189.516,Z 508.462,A -85,B 0,C 180,E1 -23928.773,E2 -23928.773} C_VEL
LIN {X 0,Y 188.444,Z 510.536,A -85,B 0,C 180,E1 -23929.757,E2 -23929.757} C_VEL
LIN {X 0,Y 180.907,Z 518.929,A -85,B 0,C 180,E1 -23932.746,E2 -23932.746} C_VEL
LIN {X 0,Y 175.162,Z 524.523,A -85,B 0,C 180,E1 -23935.397,E2 -23935.397} C_VEL
LIN {X 0,Y 168.714,Z 530.103,A -85,B 0,C 180,E1 -23938.912,E2 -23938.912} C_VEL
LIN {X 0,Y 163.402,Z 534.051,A -85,B 0,C 180,E1 -23942.464,E2 -23942.464} C_VEL
LIN {X 0,Y 160.191,Z 536.092,A -85,B 0,C 180,E1 -23945.033,E2 -23945.033} C_VEL
LIN {X 0,Y 156.408,Z 538.143,A -85,B 0,C 180,E1 -23948.654,E2 -23948.654} C_VEL
LIN {X 0,Y 152.137,Z 539.582,A -85,B 0,C 180,E1 -23954.027,E2 -23954.027} C_VEL
LIN {X 0,Y 149.46,Z 539.444,A -85,B 0,C 180,E1 -23959.217,E2 -23959.217} C_VEL
LIN {X 0,Y 148.389,Z 538.692,A -85,B 0,C 180,E1 -23962.264,E2 -23962.264} C_VEL
LIN {X 0,Y 147.655,Z 537.486,A -85,B 0,C 180,E1 -23965.364,E2 -23965.364} C_VEL
LIN {X 0,Y 147.191,Z 534.163,A -85,B 0,C 180,E1 -23970.735,E2 -23970.735} C_VEL
LIN {X 0,Y 147.577,Z 529.411,A -85,B 0,C 180,E1 -23975.936,E2 -23975.936} C_VEL
LIN {X 0,Y 148.157,Z 525.135,A -85,B 0,C 180,E1 -23979.448,E2 -23979.448} C_VEL
LIN {X 0,Y 149.339,Z 518.255,A -85,B 0,C 180,E1 -23983.958,E2 -23983.958} C_VEL
LIN {X 0,Y 150.909,Z 509.989,A -85,B 0,C 180,E1 -23988.17,E2 -23988.17} C_VEL
LIN {X 0,Y 152.93,Z 500.846,A -85,B 0,C 180,E1 -23991.881,E2 -23991.881} C_VEL
LIN {X 0,Y 155.201,Z 490.638,A -85,B 0,C 180,E1 -23995.159,E2 -23995.159} C_VEL
LIN {X 0,Y 157.554,Z 479.761,A -85,B 0,C 180,E1 -23997.943,E2 -23997.943} C_VEL
LIN {X 0,Y 157.716,Z 476.495,A -85,B 0,C 180,E1 -23998.695,E2 -23998.695} C_VEL
LIN {X 0,Y 156.602,Z 465.19,A -85,B 0,C 180,E1 -24001.149,E2 -24001.149} C_VEL
LIN {X 0,Y 155.04,Z 452.58,A -85,B 0,C 180,E1 -24003.402,E2 -24003.402} C_VEL
LIN {X 0,Y 152.761,Z 438.407,A -85,B 0,C 180,E1 -24005.444,E2 -24005.444} C_VEL
LIN {X 0,Y 151.448,Z 431.259,A -85,B 0,C 180,E1 -24006.311,E2 -24006.311} C_VEL
LIN {X 0,Y 151.656,Z 429.209,A -85,B 0,C 180,E1 -24008.233,E2 -24008.233} C_VEL
LIN {X 0,Y 151.093,Z 425.022,A -85,B 0,C 180,E1 -24012.396,E2 -24012.396} C_VEL
LIN {X 0,Y 150.7,Z 422.829,A -85,B 0,C 180,E1 -24014.786,E2 -24014.786} C_VEL
LIN {X 0,Y 151.209,Z 425.453,A -85,B 0,C 180,E1 -24019.28,E2 -24019.28} C_VEL
LIN {X 0,Y 151.568,Z 427.133,A -85,B 0,C 180,E1 -24021.998,E2 -24021.998} C_VEL
LIN {X 0,Y 152.148,Z 430.88,A -85,B 0,C 180,E1 -24027.711,E2 -24027.711} C_VEL
LIN {X 0,Y 155.359,Z 444.844,A -85,B 0,C 180,E1 -24029.994,E2 -24029.994} C_VEL
LIN {X 0,Y 157.14,Z 454.45,A -85,B 0,C 180,E1 -24031.852,E2 -24031.852} C_VEL
LIN {X 0,Y 158.402,Z 465.641,A -85,B 0,C 180,E1 -24034.347,E2 -24034.347} C_VEL
LIN {X 0,Y 158.894,Z 475.617,A -85,B 0,C 180,E1 -24036.981,E2 -24036.981} C_VEL
LIN {X 0,Y 156.513,Z 485.247,A -85,B 0,C 180,E1 -24039.737,E2 -24039.737} C_VEL
LIN {X 0,Y 154.374,Z 492.893,A -85,B 0,C 180,E1 -24042.482,E2 -24042.482} C_VEL
LIN {X 0,Y 152.231,Z 500.718,A -85,B 0,C 180,E1 -24046.075,E2 -24046.075} C_VEL
LIN {X 0,Y 150.413,Z 507.061,A -85,B 0,C 180,E1 -24049.792,E2 -24049.792} C_VEL
LIN {X 0,Y 149.103,Z 512.043,A -85,B 0,C 180,E1 -24053.612,E2 -24053.612} C_VEL
LIN {X 0,Y 148.127,Z 516.528,A -85,B 0,C 180,E1 -24058.316,E2 -24058.316} C_VEL
LIN {X 0,Y 147.815,Z 518.656,A -85,B 0,C 180,E1 -24061.526,E2 -24061.526} C_VEL
LIN {X 0,Y 148.071,Z 520.606,A -85,B 0,C 180,E1 -24066.209,E2 -24066.209} C_VEL
LIN {X 0,Y 149.214,Z 521.155,A -85,B 0,C 180,E1 -24071.245,E2 -24071.245} C_VEL
LIN {X 0,Y 151.048,Z 520.332,A -85,B 0,C 180,E1 -24075.741,E2 -24075.741} C_VEL
LIN {X 0,Y 153.656,Z 518.134,A -85,B 0,C 180,E1 -24080.184,E2 -24080.184} C_VEL
LIN {X 0,Y 156.927,Z 514.649,A -85,B 0,C 180,E1 -24084.395,E2 -24084.395} C_VEL
LIN {X 0,Y 160.991,Z 509.615,A -85,B 0,C 180,E1 -24088.41,E2 -24088.41} C_VEL
LIN {X 0,Y 165.068,Z 504.053,A -85,B 0,C 180,E1 -24091.628,E2 -24091.628} C_VEL
LIN {X 0,Y 169.332,Z 497.492,A -85,B 0,C 180,E1 -24094.502,E2 -24094.502} C_VEL
LIN {X 0,Y 171.933,Z 493.013,A -85,B 0,C 180,E1 -24096.096,E2 -24096.096} C_VEL
LIN {X 0,Y 173.081,Z 488.567,A -85,B 0,C 180,E1 -24097.94,E2 -24097.94} C_VEL
LIN {X 0,Y 173.81,Z 480.868,A -85,B 0,C 180,E1 -24101.127,E2 -24101.127} C_VEL
LIN {X 0,Y 173.764,Z 474.969,A -85,B 0,C 180,E1 -24103.554,E2 -24103.554} C_VEL
LIN {X 0,Y 173.039,Z 469.751,A -85,B 0,C 180,E1 -24105.896,E2 -24105.896} C_VEL
LIN {X 0,Y 171.192,Z 463.751,A -85,B 0,C 180,E1 -24109.056,E2 -24109.056} C_VEL
LIN {X 0,Y 169.41,Z 459.197,A -85,B 0,C 180,E1 -24111.77,E2 -24111.77} C_VEL
LIN {X 0,Y 168.159,Z 456.235,A -85,B 0,C 180,E1 -24113.702,E2 -24113.702} C_VEL
LIN {X 0,Y 165.609,Z 451.412,A -85,B 0,C 180,E1 -24117.569,E2 -24117.569} C_VEL
LIN {X 0,Y 163.345,Z 446.962,A -85,B 0,C 180,E1 -24121.85,E2 -24121.85} C_VEL
LIN {X 0,Y 159.967,Z 443.734,A -85,B 0,C 180,E1 -24130.762,E2 -24130.762} C_VEL
LIN {X 0,Y 159.629,Z 443.415,A -85,B 0,C 180,E1 -24135.318,E2 -24135.318} C_VEL
LIN {X 0,Y 160.045,Z 444.788,A -85,B 0,C 180,E1 -24139.897,E2 -24139.897} C_VEL
LIN {X 0,Y 163.483,Z 449.897,A -85,B 0,C 180,E1 -24148.485,E2 -24148.485} C_VEL
LIN {X 0,Y 165.24,Z 453.926,A -85,B 0,C 180,E1 -24151.731,E2 -24151.731} C_VEL
